KUKA KRL data list: Inconel_dataset.dat

&ACCESS RVP1
&REL 1217
&PARAM WOPTRAJECTORYID = 2
&PARAM WOPTEMPLATENAME = WopCoreTemplatePath
&PARAM DISKPATH = KRC:\R1\Program\Working Paths
DEFDAT  Inconel_dataset
;FOLD EXTERNAL DECLARATIONS;%{PE}%MKUKATPBASIS,%CEXT,%VCOMMON,%P
;FOLD BASISTECH EXT;%{PE}%MKUKATPBASIS,%CEXT,%VEXT,%P
EXT  BAS (BAS_COMMAND  :IN,REAL  :IN )
DECL INT SUCCESS
;ENDFOLD (BASISTECH EXT)
;FOLD USER EXT;%{E}%MKUKATPUSER,%CEXT,%VEXT,%P
;Make your modifications here

;ENDFOLD (USER EXT)
;ENDFOLD (EXTERNAL DECLARATIONS)

INT APP_GENNUMBER = 215375
INT APP_ANSWER
INT APP_OFFSET
DECL STATE_T APP_STATE

DECL PDAT PPDATP0={VEL 100,ACC 100,APO_DIST 5,APO_MODE #CDIS,GEAR_JERK 100.0,EXAX_IGN 0}
DECL FDAT FP0={TOOL_NO 2,BASE_NO 10,IPO_FRAME #BASE,POINT2[] " ",TQ_STATE FALSE}
DECL E6AXIS XP0={A1 -1000.000,A2 -90.000,A3 90.000,A4 0.000,A5 -90.000,A6 0.000,E1 0.000,E2 -41.000,E3 33.000,E4 0.000,E5 0.000,E6 0.000}

; Data for Routine_0
DECL LDAT LCPDATP1={VEL 1.0,ACC 100,APO_DIST 5,APO_FAC 50.0,ORI_TYP #VAR,CIRC_TYP #BASE,JERK_FAC 50.0}
DECL FDAT FP1={TOOL_NO 2,BASE_NO 10,IPO_FRAME #BASE,POINT2[] " ",TQ_STATE FALSE}
DECL E6POS XP1={X 100.000,Y 0.000,Z -100.000,A 0.000,B 0.000,C 0.000}
DECL LDAT LCPDATP2={VEL 0.116,ACC 100,APO_DIST 5,APO_FAC 50.0,ORI_TYP #VAR,CIRC_TYP #BASE,JERK_FAC 50.0}
DECL FDAT FP2={TOOL_NO 2,BASE_NO 10,IPO_FRAME #BASE,POINT2[] " ",TQ_STATE FALSE}
DECL E6POS XP2={X 50.000,Y -5.730,Z -30.020,A 0.000,B 0.000,C -28.000}
DECL LDAT LCPDATP3={VEL 0.116,ACC 100,APO_DIST 5,APO_FAC 50.0,ORI_TYP #VAR,CIRC_TYP #BASE,JERK_FAC 50.0}
DECL FDAT FP3={TOOL_NO 2,BASE_NO 10,IPO_FRAME #BASE,POINT2[] " ",TQ_STATE FALSE}
DECL E6POS XP3={X 0.000,Y -5.730,Z -30.020,A 0.000,B 0.000,C -28.000}
DECL LDAT LCPDATP4={VEL 0.116,ACC 100,APO_DIST 5,APO_FAC 50.0,ORI_TYP #VAR,CIRC_TYP #BASE,JERK_FAC 50.0}
DECL FDAT FP4={TOOL_NO 2,BASE_NO 10,IPO_FRAME #BASE,POINT2[] " ",TQ_STATE FALSE}
DECL E6POS XP4={X -50.000,Y -5.730,Z -30.020,A 0.000,B 0.000,C -28.000}
DECL LDAT LCPDATP5={VEL 0.116,ACC 100,APO_DIST 5,APO_FAC 50.0,ORI_TYP #VAR,CIRC_TYP #BASE,JERK_FAC 50.0}
DECL FDAT FP5={TOOL_NO 2,BASE_NO 10,IPO_FRAME #BASE,POINT2[] " ",TQ_STATE FALSE}
DECL E6POS XP5={X -100.000,Y -5.730,Z -30.020,A 0.000,B 0.000,C -28.000}
DECL LDAT LCPDATP6={VEL 0.099,ACC 100,APO_DIST 5,APO_FAC 50.0,ORI_TYP #VAR,CIRC_TYP #BASE,JERK_FAC 50.0}
DECL FDAT FP6={TOOL_NO 2,BASE_NO 10,IPO_FRAME #BASE,POINT2[] " ",TQ_STATE FALSE}
DECL E6POS XP6={X -100.000,Y 4.550,Z -24.510,A 0.000,B 0.000,C -40.000}
DECL LDAT LCPDATP7={VEL 0.099,ACC 100,APO_DIST 5,APO_FAC 50.0,ORI_TYP #VAR,CIRC_TYP #BASE,JERK_FAC 50.0}
DECL FDAT FP7={TOOL_NO 2,BASE_NO 10,IPO_FRAME #BASE,POINT2[] " ",TQ_STATE FALSE}
DECL E6POS XP7={X -50.000,Y 4.550,Z -24.510,A 0.000,B 0.000,C -40.000}
DECL LDAT LCPDATP8={VEL 0.099,ACC 100,APO_DIST 5,APO_FAC 50.0,ORI_TYP #VAR,CIRC_TYP #BASE,JERK_FAC 50.0}
DECL FDAT FP8={TOOL_NO 2,BASE_NO 10,IPO_FRAME #BASE,POINT2[] " ",TQ_STATE FALSE}
DECL E6POS XP8={X -0.000,Y 4.550,Z -24.510,A 0.000,B 0.000,C -40.000}
DECL LDAT LCPDATP9={VEL 0.099,ACC 100,APO_DIST 5,APO_FAC 50.0,ORI_TYP #VAR,CIRC_TYP #BASE,JERK_FAC 50.0}
DECL FDAT FP9={TOOL_NO 2,BASE_NO 10,IPO_FRAME #BASE,POINT2[] " ",TQ_STATE FALSE}
DECL E6POS XP9={X 50.000,Y 4.550,Z -24.510,A 0.000,B 0.000,C -40.000}
DECL LDAT LCPDATP10={VEL 0.075,ACC 100,APO_DIST 5,APO_FAC 50.0,ORI_TYP #VAR,CIRC_TYP #BASE,JERK_FAC 50.0}
DECL FDAT FP10={TOOL_NO 2,BASE_NO 10,IPO_FRAME #BASE,POINT2[] " ",TQ_STATE FALSE}
DECL E6POS XP10={X 50.000,Y 24.940,Z -36.820,A 0.000,B 0.000,C -23.000}
DECL LDAT LCPDATP11={VEL 0.075,ACC 100,APO_DIST 5,APO_FAC 50.0,ORI_TYP #VAR,CIRC_TYP #BASE,JERK_FAC 50.0}
DECL FDAT FP11={TOOL_NO 2,BASE_NO 10,IPO_FRAME #BASE,POINT2[] " ",TQ_STATE FALSE}
DECL E6POS XP11={X -0.000,Y 24.940,Z -36.820,A 0.000,B 0.000,C -23.000}
DECL LDAT LCPDATP12={VEL 0.075,ACC 100,APO_DIST 5,APO_FAC 50.0,ORI_TYP #VAR,CIRC_TYP #BASE,JERK_FAC 50.0}
DECL FDAT FP12={TOOL_NO 2,BASE_NO 10,IPO_FRAME #BASE,POINT2[] " ",TQ_STATE FALSE}
DECL E6POS XP12={X -50.000,Y 24.940,Z -36.820,A 0.000,B 0.000,C -23.000}
DECL LDAT LCPDATP13={VEL 0.075,ACC 100,APO_DIST 5,APO_FAC 50.0,ORI_TYP #VAR,CIRC_TYP #BASE,JERK_FAC 50.0}
DECL FDAT FP13={TOOL_NO 2,BASE_NO 10,IPO_FRAME #BASE,POINT2[] " ",TQ_STATE FALSE}
DECL E6POS XP13={X -100.000,Y 24.940,Z -36.820,A 0.000,B 0.000,C -23.000}
DECL LDAT LCPDATP14={VEL 0.113,ACC 100,APO_DIST 5,APO_FAC 50.0,ORI_TYP #VAR,CIRC_TYP #BASE,JERK_FAC 50.0}
DECL FDAT FP14={TOOL_NO 2,BASE_NO 10,IPO_FRAME #BASE,POINT2[] " ",TQ_STATE FALSE}
DECL E6POS XP14={X -100.000,Y 52.180,Z -87.790,A 0.000,B 0.000,C -4.000}
DECL LDAT LCPDATP15={VEL 0.113,ACC 100,APO_DIST 5,APO_FAC 50.0,ORI_TYP #VAR,CIRC_TYP #BASE,JERK_FAC 50.0}
DECL FDAT FP15={TOOL_NO 2,BASE_NO 10,IPO_FRAME #BASE,POINT2[] " ",TQ_STATE FALSE}
DECL E6POS XP15={X -50.000,Y 52.180,Z -87.790,A 0.000,B 0.000,C -4.000}
DECL LDAT LCPDATP16={VEL 0.113,ACC 100,APO_DIST 5,APO_FAC 50.0,ORI_TYP #VAR,CIRC_TYP #BASE,JERK_FAC 50.0}
DECL FDAT FP16={TOOL_NO 2,BASE_NO 10,IPO_FRAME #BASE,POINT2[] " ",TQ_STATE FALSE}
DECL E6POS XP16={X -0.000,Y 52.180,Z -87.790,A 0.000,B 0.000,C -4.000}
DECL LDAT LCPDATP17={VEL 0.113,ACC 100,APO_DIST 5,APO_FAC 50.0,ORI_TYP #VAR,CIRC_TYP #BASE,JERK_FAC 50.0}
DECL FDAT FP17={TOOL_NO 2,BASE_NO 10,IPO_FRAME #BASE,POINT2[] " ",TQ_STATE FALSE}
DECL E6POS XP17={X 50.000,Y 52.180,Z -87.790,A 0.000,B 0.000,C -4.000}
DECL LDAT LCPDATP18={VEL 0.086,ACC 100,APO_DIST 5,APO_FAC 50.0,ORI_TYP #VAR,CIRC_TYP #BASE,JERK_FAC 50.0}
DECL FDAT FP18={TOOL_NO 2,BASE_NO 10,IPO_FRAME #BASE,POINT2[] " ",TQ_STATE FALSE}
DECL E6POS XP18={X 50.000,Y 68.620,Z -69.900,A 0.000,B 0.000,C -3.000}
DECL LDAT LCPDATP19={VEL 0.086,ACC 100,APO_DIST 5,APO_FAC 50.0,ORI_TYP #VAR,CIRC_TYP #BASE,JERK_FAC 50.0}
DECL FDAT FP19={TOOL_NO 2,BASE_NO 10,IPO_FRAME #BASE,POINT2[] " ",TQ_STATE FALSE}
DECL E6POS XP19={X -0.000,Y 68.620,Z -69.900,A 0.000,B 0.000,C -3.000}
DECL LDAT LCPDATP20={VEL 0.086,ACC 100,APO_DIST 5,APO_FAC 50.0,ORI_TYP #VAR,CIRC_TYP #BASE,JERK_FAC 50.0}
DECL FDAT FP20={TOOL_NO 2,BASE_NO 10,IPO_FRAME #BASE,POINT2[] " ",TQ_STATE FALSE}
DECL E6POS XP20={X -50.000,Y 68.620,Z -69.900,A 0.000,B 0.000,C -3.000}
DECL LDAT LCPDATP21={VEL 0.086,ACC 100,APO_DIST 5,APO_FAC 50.0,ORI_TYP #VAR,CIRC_TYP #BASE,JERK_FAC 50.0}
DECL FDAT FP21={TOOL_NO 2,BASE_NO 10,IPO_FRAME #BASE,POINT2[] " ",TQ_STATE FALSE}
DECL E6POS XP21={X -100.000,Y 68.620,Z -69.900,A 0.000,B 0.000,C -3.000}
DECL LDAT LCPDATP22={VEL 0.073,ACC 100,APO_DIST 5,APO_FAC 50.0,ORI_TYP #VAR,CIRC_TYP #BASE,JERK_FAC 50.0}
DECL FDAT FP22={TOOL_NO 2,BASE_NO 10,IPO_FRAME #BASE,POINT2[] " ",TQ_STATE FALSE}
DECL E6POS XP22={X -100.000,Y 65.180,Z -95.090,A 0.000,B 0.000,C -14.000}
DECL LDAT LCPDATP23={VEL 0.073,ACC 100,APO_DIST 5,APO_FAC 50.0,ORI_TYP #VAR,CIRC_TYP #BASE,JERK_FAC 50.0}
DECL FDAT FP23={TOOL_NO 2,BASE_NO 10,IPO_FRAME #BASE,POINT2[] " ",TQ_STATE FALSE}
DECL E6POS XP23={X -50.000,Y 65.180,Z -95.090,A 0.000,B 0.000,C -14.000}
DECL LDAT LCPDATP24={VEL 0.073,ACC 100,APO_DIST 5,APO_FAC 50.0,ORI_TYP #VAR,CIRC_TYP #BASE,JERK_FAC 50.0}
DECL FDAT FP24={TOOL_NO 2,BASE_NO 10,IPO_FRAME #BASE,POINT2[] " ",TQ_STATE FALSE}
DECL E6POS XP24={X -0.000,Y 65.180,Z -95.090,A 0.000,B 0.000,C -14.000}
DECL LDAT LCPDATP25={VEL 0.073,ACC 100,APO_DIST 5,APO_FAC 50.0,ORI_TYP #VAR,CIRC_TYP #BASE,JERK_FAC 50.0}
DECL FDAT FP25={TOOL_NO 2,BASE_NO 10,IPO_FRAME #BASE,POINT2[] " ",TQ_STATE FALSE}
DECL E6POS XP25={X 50.000,Y 65.180,Z -95.090,A 0.000,B 0.000,C -14.000}
DECL LDAT LCPDATP26={VEL 0.137,ACC 100,APO_DIST 5,APO_FAC 50.0,ORI_TYP #VAR,CIRC_TYP #BASE,JERK_FAC 50.0}
DECL FDAT FP26={TOOL_NO 2,BASE_NO 10,IPO_FRAME #BASE,POINT2[] " ",TQ_STATE FALSE}
DECL E6POS XP26={X 50.000,Y 48.190,Z -79.460,A 0.000,B 0.000,C -35.000}
DECL LDAT LCPDATP27={VEL 0.137,ACC 100,APO_DIST 5,APO_FAC 50.0,ORI_TYP #VAR,CIRC_TYP #BASE,JERK_FAC 50.0}
DECL FDAT FP27={TOOL_NO 2,BASE_NO 10,IPO_FRAME #BASE,POINT2[] " ",TQ_STATE FALSE}
DECL E6POS XP27={X -0.000,Y 48.190,Z -79.460,A 0.000,B 0.000,C -35.000}
DECL LDAT LCPDATP28={VEL 0.137,ACC 100,APO_DIST 5,APO_FAC 50.0,ORI_TYP #VAR,CIRC_TYP #BASE,JERK_FAC 50.0}
DECL FDAT FP28={TOOL_NO 2,BASE_NO 10,IPO_FRAME #BASE,POINT2[] " ",TQ_STATE FALSE}
DECL E6POS XP28={X -50.000,Y 48.190,Z -79.460,A 0.000,B 0.000,C -35.000}
DECL LDAT LCPDATP29={VEL 0.137,ACC 100,APO_DIST 5,APO_FAC 50.0,ORI_TYP #VAR,CIRC_TYP #BASE,JERK_FAC 50.0}
DECL FDAT FP29={TOOL_NO 2,BASE_NO 10,IPO_FRAME #BASE,POINT2[] " ",TQ_STATE FALSE}
DECL E6POS XP29={X -100.000,Y 48.190,Z -79.460,A 0.000,B 0.000,C -35.000}
DECL LDAT LCPDATP30={VEL 0.082,ACC 100,APO_DIST 5,APO_FAC 50.0,ORI_TYP #VAR,CIRC_TYP #BASE,JERK_FAC 50.0}
DECL FDAT FP30={TOOL_NO 2,BASE_NO 10,IPO_FRAME #BASE,POINT2[] " ",TQ_STATE FALSE}
DECL E6POS XP30={X -100.000,Y 87.280,Z -46.640,A 0.000,B 0.000,C -32.000}
DECL LDAT LCPDATP31={VEL 0.082,ACC 100,APO_DIST 5,APO_FAC 50.0,ORI_TYP #VAR,CIRC_TYP #BASE,JERK_FAC 50.0}
DECL FDAT FP31={TOOL_NO 2,BASE_NO 10,IPO_FRAME #BASE,POINT2[] " ",TQ_STATE FALSE}
DECL E6POS XP31={X -50.000,Y 87.280,Z -46.640,A 0.000,B 0.000,C -32.000}
DECL LDAT LCPDATP32={VEL 0.082,ACC 100,APO_DIST 5,APO_FAC 50.0,ORI_TYP #VAR,CIRC_TYP #BASE,JERK_FAC 50.0}
DECL FDAT FP32={TOOL_NO 2,BASE_NO 10,IPO_FRAME #BASE,POINT2[] " ",TQ_STATE FALSE}
DECL E6POS XP32={X -0.000,Y 87.280,Z -46.640,A 0.000,B 0.000,C -32.000}
DECL LDAT LCPDATP33={VEL 0.082,ACC 100,APO_DIST 5,APO_FAC 50.0,ORI_TYP #VAR,CIRC_TYP #BASE,JERK_FAC 50.0}
DECL FDAT FP33={TOOL_NO 2,BASE_NO 10,IPO_FRAME #BASE,POINT2[] " ",TQ_STATE FALSE}
DECL E6POS XP33={X 50.000,Y 87.280,Z -46.640,A 0.000,B 0.000,C -32.000}
DECL LDAT LCPDATP34={VEL 0.086,ACC 100,APO_DIST 5,APO_FAC 50.0,ORI_TYP #VAR,CIRC_TYP #BASE,JERK_FAC 50.0}
DECL FDAT FP34={TOOL_NO 2,BASE_NO 10,IPO_FRAME #BASE,POINT2[] " ",TQ_STATE FALSE}
DECL E6POS XP34={X 50.000,Y 101.710,Z -93.610,A 0.000,B 0.000,C -19.000}
DECL LDAT LCPDATP35={VEL 0.086,ACC 100,APO_DIST 5,APO_FAC 50.0,ORI_TYP #VAR,CIRC_TYP #BASE,JERK_FAC 50.0}
DECL FDAT FP35={TOOL_NO 2,BASE_NO 10,IPO_FRAME #BASE,POINT2[] " ",TQ_STATE FALSE}
DECL E6POS XP35={X -0.000,Y 101.710,Z -93.610,A 0.000,B 0.000,C -19.000}
DECL LDAT LCPDATP36={VEL 0.086,ACC 100,APO_DIST 5,APO_FAC 50.0,ORI_TYP #VAR,CIRC_TYP #BASE,JERK_FAC 50.0}
DECL FDAT FP36={TOOL_NO 2,BASE_NO 10,IPO_FRAME #BASE,POINT2[] " ",TQ_STATE FALSE}
DECL E6POS XP36={X -50.000,Y 101.710,Z -93.610,A 0.000,B 0.000,C -19.000}
DECL LDAT LCPDATP37={VEL 0.086,ACC 100,APO_DIST 5,APO_FAC 50.0,ORI_TYP #VAR,CIRC_TYP #BASE,JERK_FAC 50.0}
DECL FDAT FP37={TOOL_NO 2,BASE_NO 10,IPO_FRAME #BASE,POINT2[] " ",TQ_STATE FALSE}
DECL E6POS XP37={X -100.000,Y 101.710,Z -93.610,A 0.000,B 0.000,C -19.000}
DECL LDAT LCPDATP38={VEL 0.097,ACC 100,APO_DIST 5,APO_FAC 50.0,ORI_TYP #VAR,CIRC_TYP #BASE,JERK_FAC 50.0}
DECL FDAT FP38={TOOL_NO 2,BASE_NO 10,IPO_FRAME #BASE,POINT2[] " ",TQ_STATE FALSE}
DECL E6POS XP38={X -100.000,Y 117.680,Z -79.350,A 0.000,B 0.000,C -21.000}
DECL LDAT LCPDATP39={VEL 0.097,ACC 100,APO_DIST 5,APO_FAC 50.0,ORI_TYP #VAR,CIRC_TYP #BASE,JERK_FAC 50.0}
DECL FDAT FP39={TOOL_NO 2,BASE_NO 10,IPO_FRAME #BASE,POINT2[] " ",TQ_STATE FALSE}
DECL E6POS XP39={X -50.000,Y 117.680,Z -79.350,A 0.000,B 0.000,C -21.000}
DECL LDAT LCPDATP40={VEL 0.097,ACC 100,APO_DIST 5,APO_FAC 50.0,ORI_TYP #VAR,CIRC_TYP #BASE,JERK_FAC 50.0}
DECL FDAT FP40={TOOL_NO 2,BASE_NO 10,IPO_FRAME #BASE,POINT2[] " ",TQ_STATE FALSE}
DECL E6POS XP40={X -0.000,Y 117.680,Z -79.350,A 0.000,B 0.000,C -21.000}
DECL LDAT LCPDATP41={VEL 0.097,ACC 100,APO_DIST 5,APO_FAC 50.0,ORI_TYP #VAR,CIRC_TYP #BASE,JERK_FAC 50.0}
DECL FDAT FP41={TOOL_NO 2,BASE_NO 10,IPO_FRAME #BASE,POINT2[] " ",TQ_STATE FALSE}
DECL E6POS XP41={X 50.000,Y 117.680,Z -79.350,A 0.000,B 0.000,C -21.000}
DECL LDAT LCPDATP42={VEL 0.136,ACC 100,APO_DIST 5,APO_FAC 50.0,ORI_TYP #VAR,CIRC_TYP #BASE,JERK_FAC 50.0}
DECL FDAT FP42={TOOL_NO 2,BASE_NO 10,IPO_FRAME #BASE,POINT2[] " ",TQ_STATE FALSE}
DECL E6POS XP42={X 50.000,Y 150.480,Z -65.980,A 0.000,B 0.000,C -10.000}
DECL LDAT LCPDATP43={VEL 0.136,ACC 100,APO_DIST 5,APO_FAC 50.0,ORI_TYP #VAR,CIRC_TYP #BASE,JERK_FAC 50.0}
DECL FDAT FP43={TOOL_NO 2,BASE_NO 10,IPO_FRAME #BASE,POINT2[] " ",TQ_STATE FALSE}
DECL E6POS XP43={X -0.000,Y 150.480,Z -65.980,A 0.000,B 0.000,C -10.000}
DECL LDAT LCPDATP44={VEL 0.136,ACC 100,APO_DIST 5,APO_FAC 50.0,ORI_TYP #VAR,CIRC_TYP #BASE,JERK_FAC 50.0}
DECL FDAT FP44={TOOL_NO 2,BASE_NO 10,IPO_FRAME #BASE,POINT2[] " ",TQ_STATE FALSE}
DECL E6POS XP44={X -50.000,Y 150.480,Z -65.980,A 0.000,B 0.000,C -10.000}
DECL LDAT LCPDATP45={VEL 0.136,ACC 100,APO_DIST 5,APO_FAC 50.0,ORI_TYP #VAR,CIRC_TYP #BASE,JERK_FAC 50.0}
DECL FDAT FP45={TOOL_NO 2,BASE_NO 10,IPO_FRAME #BASE,POINT2[] " ",TQ_STATE FALSE}
DECL E6POS XP45={X -100.000,Y 150.480,Z -65.980,A 0.000,B 0.000,C -10.000}
DECL LDAT LCPDATP46={VEL 0.107,ACC 100,APO_DIST 5,APO_FAC 50.0,ORI_TYP #VAR,CIRC_TYP #BASE,JERK_FAC 50.0}
DECL FDAT FP46={TOOL_NO 2,BASE_NO 10,IPO_FRAME #BASE,POINT2[] " ",TQ_STATE FALSE}
DECL E6POS XP46={X -100.000,Y 132.510,Z -57.520,A 0.000,B 0.000,C -38.000}
DECL LDAT LCPDATP47={VEL 0.107,ACC 100,APO_DIST 5,APO_FAC 50.0,ORI_TYP #VAR,CIRC_TYP #BASE,JERK_FAC 50.0}
DECL FDAT FP47={TOOL_NO 2,BASE_NO 10,IPO_FRAME #BASE,POINT2[] " ",TQ_STATE FALSE}
DECL E6POS XP47={X -50.000,Y 132.510,Z -57.520,A 0.000,B 0.000,C -38.000}
DECL LDAT LCPDATP48={VEL 0.107,ACC 100,APO_DIST 5,APO_FAC 50.0,ORI_TYP #VAR,CIRC_TYP #BASE,JERK_FAC 50.0}
DECL FDAT FP48={TOOL_NO 2,BASE_NO 10,IPO_FRAME #BASE,POINT2[] " ",TQ_STATE FALSE}
DECL E6POS XP48={X -0.000,Y 132.510,Z -57.520,A 0.000,B 0.000,C -38.000}
DECL LDAT LCPDATP49={VEL 0.107,ACC 100,APO_DIST 5,APO_FAC 50.0,ORI_TYP #VAR,CIRC_TYP #BASE,JERK_FAC 50.0}
DECL FDAT FP49={TOOL_NO 2,BASE_NO 10,IPO_FRAME #BASE,POINT2[] " ",TQ_STATE FALSE}
DECL E6POS XP49={X 50.000,Y 132.510,Z -57.520,A 0.000,B 0.000,C -38.000}
DECL LDAT LCPDATP50={VEL 0.09,ACC 100,APO_DIST 5,APO_FAC 50.0,ORI_TYP #VAR,CIRC_TYP #BASE,JERK_FAC 50.0}
DECL FDAT FP50={TOOL_NO 2,BASE_NO 10,IPO_FRAME #BASE,POINT2[] " ",TQ_STATE FALSE}
DECL E6POS XP50={X 50.000,Y 148.310,Z -68.770,A 0.000,B 0.000,C -33.000}
DECL LDAT LCPDATP51={VEL 0.09,ACC 100,APO_DIST 5,APO_FAC 50.0,ORI_TYP #VAR,CIRC_TYP #BASE,JERK_FAC 50.0}
DECL FDAT FP51={TOOL_NO 2,BASE_NO 10,IPO_FRAME #BASE,POINT2[] " ",TQ_STATE FALSE}
DECL E6POS XP51={X -0.000,Y 148.310,Z -68.770,A 0.000,B 0.000,C -33.000}
DECL LDAT LCPDATP52={VEL 0.09,ACC 100,APO_DIST 5,APO_FAC 50.0,ORI_TYP #VAR,CIRC_TYP #BASE,JERK_FAC 50.0}
DECL FDAT FP52={TOOL_NO 2,BASE_NO 10,IPO_FRAME #BASE,POINT2[] " ",TQ_STATE FALSE}
DECL E6POS XP52={X -50.000,Y 148.310,Z -68.770,A 0.000,B 0.000,C -33.000}
DECL LDAT LCPDATP53={VEL 0.09,ACC 100,APO_DIST 5,APO_FAC 50.0,ORI_TYP #VAR,CIRC_TYP #BASE,JERK_FAC 50.0}
DECL FDAT FP53={TOOL_NO 2,BASE_NO 10,IPO_FRAME #BASE,POINT2[] " ",TQ_STATE FALSE}
DECL E6POS XP53={X -100.000,Y 148.310,Z -68.770,A 0.000,B 0.000,C -33.000}
DECL LDAT LCPDATP54={VEL 0.132,ACC 100,APO_DIST 5,APO_FAC 50.0,ORI_TYP #VAR,CIRC_TYP #BASE,JERK_FAC 50.0}
DECL FDAT FP54={TOOL_NO 2,BASE_NO 10,IPO_FRAME #BASE,POINT2[] " ",TQ_STATE FALSE}
DECL E6POS XP54={X -100.000,Y 203.750,Z -95.870,A 0.000,B 0.000,C -3.000}
DECL LDAT LCPDATP55={VEL 0.132,ACC 100,APO_DIST 5,APO_FAC 50.0,ORI_TYP #VAR,CIRC_TYP #BASE,JERK_FAC 50.0}
DECL FDAT FP55={TOOL_NO 2,BASE_NO 10,IPO_FRAME #BASE,POINT2[] " ",TQ_STATE FALSE}
DECL E6POS XP55={X -50.000,Y 203.750,Z -95.870,A 0.000,B 0.000,C -3.000}
DECL LDAT LCPDATP56={VEL 0.132,ACC 100,APO_DIST 5,APO_FAC 50.0,ORI_TYP #VAR,CIRC_TYP #BASE,JERK_FAC 50.0}
DECL FDAT FP56={TOOL_NO 2,BASE_NO 10,IPO_FRAME #BASE,POINT2[] " ",TQ_STATE FALSE}
DECL E6POS XP56={X -0.000,Y 203.750,Z -95.870,A 0.000,B 0.000,C -3.000}
DECL LDAT LCPDATP57={VEL 0.132,ACC 100,APO_DIST 5,APO_FAC 50.0,ORI_TYP #VAR,CIRC_TYP #BASE,JERK_FAC 50.0}
DECL FDAT FP57={TOOL_NO 2,BASE_NO 10,IPO_FRAME #BASE,POINT2[] " ",TQ_STATE FALSE}
DECL E6POS XP57={X 50.000,Y 203.750,Z -95.870,A 0.000,B 0.000,C -3.000}
DECL LDAT LCPDATP58={VEL 0.068,ACC 100,APO_DIST 5,APO_FAC 50.0,ORI_TYP #VAR,CIRC_TYP #BASE,JERK_FAC 50.0}
DECL FDAT FP58={TOOL_NO 2,BASE_NO 10,IPO_FRAME #BASE,POINT2[] " ",TQ_STATE FALSE}
DECL E6POS XP58={X 50.000,Y 221.500,Z -80.990,A 0.000,B 0.000,C -1.000}
DECL LDAT LCPDATP59={VEL 0.068,ACC 100,APO_DIST 5,APO_FAC 50.0,ORI_TYP #VAR,CIRC_TYP #BASE,JERK_FAC 50.0}
DECL FDAT FP59={TOOL_NO 2,BASE_NO 10,IPO_FRAME #BASE,POINT2[] " ",TQ_STATE FALSE}
DECL E6POS XP59={X -0.000,Y 221.500,Z -80.990,A 0.000,B 0.000,C -1.000}
DECL LDAT LCPDATP60={VEL 0.068,ACC 100,APO_DIST 5,APO_FAC 50.0,ORI_TYP #VAR,CIRC_TYP #BASE,JERK_FAC 50.0}
DECL FDAT FP60={TOOL_NO 2,BASE_NO 10,IPO_FRAME #BASE,POINT2[] " ",TQ_STATE FALSE}
DECL E6POS XP60={X -50.000,Y 221.500,Z -80.990,A 0.000,B 0.000,C -1.000}
DECL LDAT LCPDATP61={VEL 0.068,ACC 100,APO_DIST 5,APO_FAC 50.0,ORI_TYP #VAR,CIRC_TYP #BASE,JERK_FAC 50.0}
DECL FDAT FP61={TOOL_NO 2,BASE_NO 10,IPO_FRAME #BASE,POINT2[] " ",TQ_STATE FALSE}
DECL E6POS XP61={X -100.000,Y 221.500,Z -80.990,A 0.000,B 0.000,C -1.000}
DECL LDAT LCPDATP62={VEL 0.115,ACC 100,APO_DIST 5,APO_FAC 50.0,ORI_TYP #VAR,CIRC_TYP #BASE,JERK_FAC 50.0}
DECL FDAT FP62={TOOL_NO 2,BASE_NO 10,IPO_FRAME #BASE,POINT2[] " ",TQ_STATE FALSE}
DECL E6POS XP62={X -100.000,Y 206.270,Z -52.830,A 0.000,B 0.000,C -30.000}
DECL LDAT LCPDATP63={VEL 0.115,ACC 100,APO_DIST 5,APO_FAC 50.0,ORI_TYP #VAR,CIRC_TYP #BASE,JERK_FAC 50.0}
DECL FDAT FP63={TOOL_NO 2,BASE_NO 10,IPO_FRAME #BASE,POINT2[] " ",TQ_STATE FALSE}
DECL E6POS XP63={X -50.000,Y 206.270,Z -52.830,A 0.000,B 0.000,C -30.000}
DECL LDAT LCPDATP64={VEL 0.115,ACC 100,APO_DIST 5,APO_FAC 50.0,ORI_TYP #VAR,CIRC_TYP #BASE,JERK_FAC 50.0}
DECL FDAT FP64={TOOL_NO 2,BASE_NO 10,IPO_FRAME #BASE,POINT2[] " ",TQ_STATE FALSE}
DECL E6POS XP64={X -0.000,Y 206.270,Z -52.830,A 0.000,B 0.000,C -30.000}
DECL LDAT LCPDATP65={VEL 0.115,ACC 100,APO_DIST 5,APO_FAC 50.0,ORI_TYP #VAR,CIRC_TYP #BASE,JERK_FAC 50.0}
DECL FDAT FP65={TOOL_NO 2,BASE_NO 10,IPO_FRAME #BASE,POINT2[] " ",TQ_STATE FALSE}
DECL E6POS XP65={X 50.000,Y 206.270,Z -52.830,A 0.000,B 0.000,C -30.000}
DECL LDAT LCPDATP66={VEL 0.111,ACC 100,APO_DIST 5,APO_FAC 50.0,ORI_TYP #VAR,CIRC_TYP #BASE,JERK_FAC 50.0}
DECL FDAT FP66={TOOL_NO 2,BASE_NO 10,IPO_FRAME #BASE,POINT2[] " ",TQ_STATE FALSE}
DECL E6POS XP66={X 50.000,Y 214.030,Z -89.530,A 0.000,B 0.000,C -24.000}
DECL LDAT LCPDATP67={VEL 0.111,ACC 100,APO_DIST 5,APO_FAC 50.0,ORI_TYP #VAR,CIRC_TYP #BASE,JERK_FAC 50.0}
DECL FDAT FP67={TOOL_NO 2,BASE_NO 10,IPO_FRAME #BASE,POINT2[] " ",TQ_STATE FALSE}
DECL E6POS XP67={X -0.000,Y 214.030,Z -89.530,A 0.000,B 0.000,C -24.000}
DECL LDAT LCPDATP68={VEL 0.111,ACC 100,APO_DIST 5,APO_FAC 50.0,ORI_TYP #VAR,CIRC_TYP #BASE,JERK_FAC 50.0}
DECL FDAT FP68={TOOL_NO 2,BASE_NO 10,IPO_FRAME #BASE,POINT2[] " ",TQ_STATE FALSE}
DECL E6POS XP68={X -50.000,Y 214.030,Z -89.530,A 0.000,B 0.000,C -24.000}
DECL LDAT LCPDATP69={VEL 0.111,ACC 100,APO_DIST 5,APO_FAC 50.0,ORI_TYP #VAR,CIRC_TYP #BASE,JERK_FAC 50.0}
DECL FDAT FP69={TOOL_NO 2,BASE_NO 10,IPO_FRAME #BASE,POINT2[] " ",TQ_STATE FALSE}
DECL E6POS XP69={X -100.000,Y 214.030,Z -89.530,A 0.000,B 0.000,C -24.000}
DECL LDAT LCPDATP70={VEL 0.124,ACC 100,APO_DIST 5,APO_FAC 50.0,ORI_TYP #VAR,CIRC_TYP #BASE,JERK_FAC 50.0}
DECL FDAT FP70={TOOL_NO 2,BASE_NO 10,IPO_FRAME #BASE,POINT2[] " ",TQ_STATE FALSE}
DECL E6POS XP70={X -100.000,Y 264.220,Z -41.970,A 0.000,B 0.000,C -2.000}
DECL LDAT LCPDATP71={VEL 0.124,ACC 100,APO_DIST 5,APO_FAC 50.0,ORI_TYP #VAR,CIRC_TYP #BASE,JERK_FAC 50.0}
DECL FDAT FP71={TOOL_NO 2,BASE_NO 10,IPO_FRAME #BASE,POINT2[] " ",TQ_STATE FALSE}
DECL E6POS XP71={X -50.000,Y 264.220,Z -41.970,A 0.000,B 0.000,C -2.000}
DECL LDAT LCPDATP72={VEL 0.124,ACC 100,APO_DIST 5,APO_FAC 50.0,ORI_TYP #VAR,CIRC_TYP #BASE,JERK_FAC 50.0}
DECL FDAT FP72={TOOL_NO 2,BASE_NO 10,IPO_FRAME #BASE,POINT2[] " ",TQ_STATE FALSE}
DECL E6POS XP72={X -0.000,Y 264.220,Z -41.970,A 0.000,B 0.000,C -2.000}
DECL LDAT LCPDATP73={VEL 0.124,ACC 100,APO_DIST 5,APO_FAC 50.0,ORI_TYP #VAR,CIRC_TYP #BASE,JERK_FAC 50.0}
DECL FDAT FP73={TOOL_NO 2,BASE_NO 10,IPO_FRAME #BASE,POINT2[] " ",TQ_STATE FALSE}
DECL E6POS XP73={X 50.000,Y 264.220,Z -41.970,A 0.000,B 0.000,C -2.000}
DECL LDAT LCPDATP74={VEL 0.112,ACC 100,APO_DIST 5,APO_FAC 50.0,ORI_TYP #VAR,CIRC_TYP #BASE,JERK_FAC 50.0}
DECL FDAT FP74={TOOL_NO 2,BASE_NO 10,IPO_FRAME #BASE,POINT2[] " ",TQ_STATE FALSE}
DECL E6POS XP74={X 50.000,Y 254.510,Z -62.120,A 0.000,B 0.000,C -24.000}
DECL LDAT LCPDATP75={VEL 0.112,ACC 100,APO_DIST 5,APO_FAC 50.0,ORI_TYP #VAR,CIRC_TYP #BASE,JERK_FAC 50.0}
DECL FDAT FP75={TOOL_NO 2,BASE_NO 10,IPO_FRAME #BASE,POINT2[] " ",TQ_STATE FALSE}
DECL E6POS XP75={X -0.000,Y 254.510,Z -62.120,A 0.000,B 0.000,C -24.000}
DECL LDAT LCPDATP76={VEL 0.112,ACC 100,APO_DIST 5,APO_FAC 50.0,ORI_TYP #VAR,CIRC_TYP #BASE,JERK_FAC 50.0}
DECL FDAT FP76={TOOL_NO 2,BASE_NO 10,IPO_FRAME #BASE,POINT2[] " ",TQ_STATE FALSE}
DECL E6POS XP76={X -50.000,Y 254.510,Z -62.120,A 0.000,B 0.000,C -24.000}
DECL LDAT LCPDATP77={VEL 0.112,ACC 100,APO_DIST 5,APO_FAC 50.0,ORI_TYP #VAR,CIRC_TYP #BASE,JERK_FAC 50.0}
DECL FDAT FP77={TOOL_NO 2,BASE_NO 10,IPO_FRAME #BASE,POINT2[] " ",TQ_STATE FALSE}
DECL E6POS XP77={X -100.000,Y 254.510,Z -62.120,A 0.000,B 0.000,C -24.000}
DECL LDAT LCPDATP78={VEL 0.109,ACC 100,APO_DIST 5,APO_FAC 50.0,ORI_TYP #VAR,CIRC_TYP #BASE,JERK_FAC 50.0}
DECL FDAT FP78={TOOL_NO 2,BASE_NO 10,IPO_FRAME #BASE,POINT2[] " ",TQ_STATE FALSE}
DECL E6POS XP78={X -100.000,Y 269.410,Z -36.410,A 0.000,B 0.000,C -36.000}
DECL LDAT LCPDATP79={VEL 0.109,ACC 100,APO_DIST 5,APO_FAC 50.0,ORI_TYP #VAR,CIRC_TYP #BASE,JERK_FAC 50.0}
DECL FDAT FP79={TOOL_NO 2,BASE_NO 10,IPO_FRAME #BASE,POINT2[] " ",TQ_STATE FALSE}
DECL E6POS XP79={X -50.000,Y 269.410,Z -36.410,A 0.000,B 0.000,C -36.000}
DECL LDAT LCPDATP80={VEL 0.109,ACC 100,APO_DIST 5,APO_FAC 50.0,ORI_TYP #VAR,CIRC_TYP #BASE,JERK_FAC 50.0}
DECL FDAT FP80={TOOL_NO 2,BASE_NO 10,IPO_FRAME #BASE,POINT2[] " ",TQ_STATE FALSE}
DECL E6POS XP80={X -0.000,Y 269.410,Z -36.410,A 0.000,B 0.000,C -36.000}
DECL LDAT LCPDATP81={VEL 0.109,ACC 100,APO_DIST 5,APO_FAC 50.0,ORI_TYP #VAR,CIRC_TYP #BASE,JERK_FAC 50.0}
DECL FDAT FP81={TOOL_NO 2,BASE_NO 10,IPO_FRAME #BASE,POINT2[] " ",TQ_STATE FALSE}
DECL E6POS XP81={X 50.000,Y 269.410,Z -36.410,A 0.000,B 0.000,C -36.000}
DECL LDAT LCPDATP82={VEL 0.104,ACC 100,APO_DIST 5,APO_FAC 50.0,ORI_TYP #VAR,CIRC_TYP #BASE,JERK_FAC 50.0}
DECL FDAT FP82={TOOL_NO 2,BASE_NO 10,IPO_FRAME #BASE,POINT2[] " ",TQ_STATE FALSE}
DECL E6POS XP82={X 50.000,Y 288.080,Z -43.260,A 0.000,B 0.000,C -28.000}
DECL LDAT LCPDATP83={VEL 0.104,ACC 100,APO_DIST 5,APO_FAC 50.0,ORI_TYP #VAR,CIRC_TYP #BASE,JERK_FAC 50.0}
DECL FDAT FP83={TOOL_NO 2,BASE_NO 10,IPO_FRAME #BASE,POINT2[] " ",TQ_STATE FALSE}
DECL E6POS XP83={X -0.000,Y 288.080,Z -43.260,A 0.000,B 0.000,C -28.000}
DECL LDAT LCPDATP84={VEL 0.104,ACC 100,APO_DIST 5,APO_FAC 50.0,ORI_TYP #VAR,CIRC_TYP #BASE,JERK_FAC 50.0}
DECL FDAT FP84={TOOL_NO 2,BASE_NO 10,IPO_FRAME #BASE,POINT2[] " ",TQ_STATE FALSE}
DECL E6POS XP84={X -50.000,Y 288.080,Z -43.260,A 0.000,B 0.000,C -28.000}
DECL LDAT LCPDATP85={VEL 0.104,ACC 100,APO_DIST 5,APO_FAC 50.0,ORI_TYP #VAR,CIRC_TYP #BASE,JERK_FAC 50.0}
DECL FDAT FP85={TOOL_NO 2,BASE_NO 10,IPO_FRAME #BASE,POINT2[] " ",TQ_STATE FALSE}
DECL E6POS XP85={X -100.000,Y 288.080,Z -43.260,A 0.000,B 0.000,C -28.000}
DECL LDAT LCPDATP86={VEL 0.053,ACC 100,APO_DIST 5,APO_FAC 50.0,ORI_TYP #VAR,CIRC_TYP #BASE,JERK_FAC 50.0}
DECL FDAT FP86={TOOL_NO 2,BASE_NO 10,IPO_FRAME #BASE,POINT2[] " ",TQ_STATE FALSE}
DECL E6POS XP86={X -100.000,Y 303.890,Z -73.230,A 0.000,B 0.000,C -18.000}
DECL LDAT LCPDATP87={VEL 0.053,ACC 100,APO_DIST 5,APO_FAC 50.0,ORI_TYP #VAR,CIRC_TYP #BASE,JERK_FAC 50.0}
DECL FDAT FP87={TOOL_NO 2,BASE_NO 10,IPO_FRAME #BASE,POINT2[] " ",TQ_STATE FALSE}
DECL E6POS XP87={X -50.000,Y 303.890,Z -73.230,A 0.000,B 0.000,C -18.000}
DECL LDAT LCPDATP88={VEL 0.053,ACC 100,APO_DIST 5,APO_FAC 50.0,ORI_TYP #VAR,CIRC_TYP #BASE,JERK_FAC 50.0}
DECL FDAT FP88={TOOL_NO 2,BASE_NO 10,IPO_FRAME #BASE,POINT2[] " ",TQ_STATE FALSE}
DECL E6POS XP88={X -0.000,Y 303.890,Z -73.230,A 0.000,B 0.000,C -18.000}
DECL LDAT LCPDATP89={VEL 0.053,ACC 100,APO_DIST 5,APO_FAC 50.0,ORI_TYP #VAR,CIRC_TYP #BASE,JERK_FAC 50.0}
DECL FDAT FP89={TOOL_NO 2,BASE_NO 10,IPO_FRAME #BASE,POINT2[] " ",TQ_STATE FALSE}
DECL E6POS XP89={X 50.000,Y 303.890,Z -73.230,A 0.000,B 0.000,C -18.000}
DECL LDAT LCPDATP90={VEL 0.063,ACC 100,APO_DIST 5,APO_FAC 50.0,ORI_TYP #VAR,CIRC_TYP #BASE,JERK_FAC 50.0}
DECL FDAT FP90={TOOL_NO 2,BASE_NO 10,IPO_FRAME #BASE,POINT2[] " ",TQ_STATE FALSE}
DECL E6POS XP90={X 50.000,Y 335.430,Z -94.640,A 0.000,B 0.000,C -5.000}
DECL LDAT LCPDATP91={VEL 0.063,ACC 100,APO_DIST 5,APO_FAC 50.0,ORI_TYP #VAR,CIRC_TYP #BASE,JERK_FAC 50.0}
DECL FDAT FP91={TOOL_NO 2,BASE_NO 10,IPO_FRAME #BASE,POINT2[] " ",TQ_STATE FALSE}
DECL E6POS XP91={X -0.000,Y 335.430,Z -94.640,A 0.000,B 0.000,C -5.000}
DECL LDAT LCPDATP92={VEL 0.063,ACC 100,APO_DIST 5,APO_FAC 50.0,ORI_TYP #VAR,CIRC_TYP #BASE,JERK_FAC 50.0}
DECL FDAT FP92={TOOL_NO 2,BASE_NO 10,IPO_FRAME #BASE,POINT2[] " ",TQ_STATE FALSE}
DECL E6POS XP92={X -50.000,Y 335.430,Z -94.640,A 0.000,B 0.000,C -5.000}
DECL LDAT LCPDATP93={VEL 0.063,ACC 100,APO_DIST 5,APO_FAC 50.0,ORI_TYP #VAR,CIRC_TYP #BASE,JERK_FAC 50.0}
DECL FDAT FP93={TOOL_NO 2,BASE_NO 10,IPO_FRAME #BASE,POINT2[] " ",TQ_STATE FALSE}
DECL E6POS XP93={X -100.000,Y 335.430,Z -94.640,A 0.000,B 0.000,C -5.000}
DECL LDAT LCPDATP94={VEL 0.5,ACC 100,APO_DIST 5,APO_FAC 50.0,ORI_TYP #VAR,CIRC_TYP #BASE,JERK_FAC 50.0}
DECL FDAT FP94={TOOL_NO 2,BASE_NO 10,IPO_FRAME #BASE,POINT2[] " ",TQ_STATE FALSE}
DECL E6POS XP94={X -150.000,Y 343.710,Z -50.000,A 0.000,B 0.000,C 0.000}
DECL LDAT LCPDATP95={VEL 1.0,ACC 100,APO_DIST 5,APO_FAC 50.0,ORI_TYP #VAR,CIRC_TYP #BASE,JERK_FAC 50.0}
DECL FDAT FP95={TOOL_NO 2,BASE_NO 10,IPO_FRAME #BASE,POINT2[] " ",TQ_STATE FALSE}
DECL E6POS XP95={X -150.000,Y 380.000,Z -20.000,A 0.000,B 0.000,C 0.000}
DECL LDAT LCPDATP96={VEL 1.0,ACC 100,APO_DIST 5,APO_FAC 50.0,ORI_TYP #VAR,CIRC_TYP #BASE,JERK_FAC 50.0}
DECL FDAT FP96={TOOL_NO 2,BASE_NO 10,IPO_FRAME #BASE,POINT2[] " ",TQ_STATE FALSE}
DECL E6POS XP96={X 100.000,Y 380.000,Z -20.000,A 0.000,B 0.000,C 0.000}
;ENDDAT for Routine_0


; Data for Routine_1
DECL LDAT LCPDATP97={VEL 1.0,ACC 100,APO_DIST 5,APO_FAC 50.0,ORI_TYP #VAR,CIRC_TYP #BASE,JERK_FAC 50.0}
DECL FDAT FP97={TOOL_NO 2,BASE_NO 9,IPO_FRAME #BASE,POINT2[] " ",TQ_STATE FALSE}
DECL E6POS XP97={X 100.000,Y 0.000,Z -100.000,A 0.000,B 0.000,C 0.000}
DECL LDAT LCPDATP98={VEL 0.065,ACC 100,APO_DIST 5,APO_FAC 50.0,ORI_TYP #VAR,CIRC_TYP #BASE,JERK_FAC 50.0}
DECL FDAT FP98={TOOL_NO 2,BASE_NO 9,IPO_FRAME #BASE,POINT2[] " ",TQ_STATE FALSE}
DECL E6POS XP98={X 50.000,Y -2.120,Z -67.490,A 0.000,B 0.000,C -12.000}
DECL LDAT LCPDATP99={VEL 0.065,ACC 100,APO_DIST 5,APO_FAC 50.0,ORI_TYP #VAR,CIRC_TYP #BASE,JERK_FAC 50.0}
DECL FDAT FP99={TOOL_NO 2,BASE_NO 9,IPO_FRAME #BASE,POINT2[] " ",TQ_STATE FALSE}
DECL E6POS XP99={X 0.000,Y -2.120,Z -67.490,A 0.000,B 0.000,C -12.000}
DECL LDAT LCPDATP100={VEL 0.065,ACC 100,APO_DIST 5,APO_FAC 50.0,ORI_TYP #VAR,CIRC_TYP #BASE,JERK_FAC 50.0}
DECL FDAT FP100={TOOL_NO 2,BASE_NO 9,IPO_FRAME #BASE,POINT2[] " ",TQ_STATE FALSE}
DECL E6POS XP100={X -50.000,Y -2.120,Z -67.490,A 0.000,B 0.000,C -12.000}
DECL LDAT LCPDATP101={VEL 0.065,ACC 100,APO_DIST 5,APO_FAC 50.0,ORI_TYP #VAR,CIRC_TYP #BASE,JERK_FAC 50.0}
DECL FDAT FP101={TOOL_NO 2,BASE_NO 9,IPO_FRAME #BASE,POINT2[] " ",TQ_STATE FALSE}
DECL E6POS XP101={X -100.000,Y -2.120,Z -67.490,A 0.000,B 0.000,C -12.000}
DECL LDAT LCPDATP102={VEL 0.088,ACC 100,APO_DIST 5,APO_FAC 50.0,ORI_TYP #VAR,CIRC_TYP #BASE,JERK_FAC 50.0}
DECL FDAT FP102={TOOL_NO 2,BASE_NO 9,IPO_FRAME #BASE,POINT2[] " ",TQ_STATE FALSE}
DECL E6POS XP102={X -100.000,Y 15.760,Z -30.600,A 0.000,B 0.000,C -17.000}
DECL LDAT LCPDATP103={VEL 0.088,ACC 100,APO_DIST 5,APO_FAC 50.0,ORI_TYP #VAR,CIRC_TYP #BASE,JERK_FAC 50.0}
DECL FDAT FP103={TOOL_NO 2,BASE_NO 9,IPO_FRAME #BASE,POINT2[] " ",TQ_STATE FALSE}
DECL E6POS XP103={X -50.000,Y 15.760,Z -30.600,A 0.000,B 0.000,C -17.000}
DECL LDAT LCPDATP104={VEL 0.088,ACC 100,APO_DIST 5,APO_FAC 50.0,ORI_TYP #VAR,CIRC_TYP #BASE,JERK_FAC 50.0}
DECL FDAT FP104={TOOL_NO 2,BASE_NO 9,IPO_FRAME #BASE,POINT2[] " ",TQ_STATE FALSE}
DECL E6POS XP104={X -0.000,Y 15.760,Z -30.600,A 0.000,B 0.000,C -17.000}
DECL LDAT LCPDATP105={VEL 0.088,ACC 100,APO_DIST 5,APO_FAC 50.0,ORI_TYP #VAR,CIRC_TYP #BASE,JERK_FAC 50.0}
DECL FDAT FP105={TOOL_NO 2,BASE_NO 9,IPO_FRAME #BASE,POINT2[] " ",TQ_STATE FALSE}
DECL E6POS XP105={X 50.000,Y 15.760,Z -30.600,A 0.000,B 0.000,C -17.000}
DECL LDAT LCPDATP106={VEL 0.06,ACC 100,APO_DIST 5,APO_FAC 50.0,ORI_TYP #VAR,CIRC_TYP #BASE,JERK_FAC 50.0}
DECL FDAT FP106={TOOL_NO 2,BASE_NO 9,IPO_FRAME #BASE,POINT2[] " ",TQ_STATE FALSE}
DECL E6POS XP106={X 50.000,Y 13.210,Z -73.250,A 0.000,B 0.000,C -22.000}
DECL LDAT LCPDATP107={VEL 0.06,ACC 100,APO_DIST 5,APO_FAC 50.0,ORI_TYP #VAR,CIRC_TYP #BASE,JERK_FAC 50.0}
DECL FDAT FP107={TOOL_NO 2,BASE_NO 9,IPO_FRAME #BASE,POINT2[] " ",TQ_STATE FALSE}
DECL E6POS XP107={X -0.000,Y 13.210,Z -73.250,A 0.000,B 0.000,C -22.000}
DECL LDAT LCPDATP108={VEL 0.06,ACC 100,APO_DIST 5,APO_FAC 50.0,ORI_TYP #VAR,CIRC_TYP #BASE,JERK_FAC 50.0}
DECL FDAT FP108={TOOL_NO 2,BASE_NO 9,IPO_FRAME #BASE,POINT2[] " ",TQ_STATE FALSE}
DECL E6POS XP108={X -50.000,Y 13.210,Z -73.250,A 0.000,B 0.000,C -22.000}
DECL LDAT LCPDATP109={VEL 0.06,ACC 100,APO_DIST 5,APO_FAC 50.0,ORI_TYP #VAR,CIRC_TYP #BASE,JERK_FAC 50.0}
DECL FDAT FP109={TOOL_NO 2,BASE_NO 9,IPO_FRAME #BASE,POINT2[] " ",TQ_STATE FALSE}
DECL E6POS XP109={X -100.000,Y 13.210,Z -73.250,A 0.000,B 0.000,C -22.000}
DECL LDAT LCPDATP110={VEL 0.135,ACC 100,APO_DIST 5,APO_FAC 50.0,ORI_TYP #VAR,CIRC_TYP #BASE,JERK_FAC 50.0}
DECL FDAT FP110={TOOL_NO 2,BASE_NO 9,IPO_FRAME #BASE,POINT2[] " ",TQ_STATE FALSE}
DECL E6POS XP110={X -100.000,Y 40.110,Z -53.550,A 0.000,B 0.000,C -17.000}
DECL LDAT LCPDATP111={VEL 0.135,ACC 100,APO_DIST 5,APO_FAC 50.0,ORI_TYP #VAR,CIRC_TYP #BASE,JERK_FAC 50.0}
DECL FDAT FP111={TOOL_NO 2,BASE_NO 9,IPO_FRAME #BASE,POINT2[] " ",TQ_STATE FALSE}
DECL E6POS XP111={X -50.000,Y 40.110,Z -53.550,A 0.000,B 0.000,C -17.000}
DECL LDAT LCPDATP112={VEL 0.135,ACC 100,APO_DIST 5,APO_FAC 50.0,ORI_TYP #VAR,CIRC_TYP #BASE,JERK_FAC 50.0}
DECL FDAT FP112={TOOL_NO 2,BASE_NO 9,IPO_FRAME #BASE,POINT2[] " ",TQ_STATE FALSE}
DECL E6POS XP112={X -0.000,Y 40.110,Z -53.550,A 0.000,B 0.000,C -17.000}
DECL LDAT LCPDATP113={VEL 0.135,ACC 100,APO_DIST 5,APO_FAC 50.0,ORI_TYP #VAR,CIRC_TYP #BASE,JERK_FAC 50.0}
DECL FDAT FP113={TOOL_NO 2,BASE_NO 9,IPO_FRAME #BASE,POINT2[] " ",TQ_STATE FALSE}
DECL E6POS XP113={X 50.000,Y 40.110,Z -53.550,A 0.000,B 0.000,C -17.000}
DECL LDAT LCPDATP114={VEL 0.119,ACC 100,APO_DIST 5,APO_FAC 50.0,ORI_TYP #VAR,CIRC_TYP #BASE,JERK_FAC 50.0}
DECL FDAT FP114={TOOL_NO 2,BASE_NO 9,IPO_FRAME #BASE,POINT2[] " ",TQ_STATE FALSE}
DECL E6POS XP114={X 50.000,Y 24.230,Z -59.840,A 0.000,B 0.000,C -39.000}
DECL LDAT LCPDATP115={VEL 0.119,ACC 100,APO_DIST 5,APO_FAC 50.0,ORI_TYP #VAR,CIRC_TYP #BASE,JERK_FAC 50.0}
DECL FDAT FP115={TOOL_NO 2,BASE_NO 9,IPO_FRAME #BASE,POINT2[] " ",TQ_STATE FALSE}
DECL E6POS XP115={X -0.000,Y 24.230,Z -59.840,A 0.000,B 0.000,C -39.000}
DECL LDAT LCPDATP116={VEL 0.119,ACC 100,APO_DIST 5,APO_FAC 50.0,ORI_TYP #VAR,CIRC_TYP #BASE,JERK_FAC 50.0}
DECL FDAT FP116={TOOL_NO 2,BASE_NO 9,IPO_FRAME #BASE,POINT2[] " ",TQ_STATE FALSE}
DECL E6POS XP116={X -50.000,Y 24.230,Z -59.840,A 0.000,B 0.000,C -39.000}
DECL LDAT LCPDATP117={VEL 0.119,ACC 100,APO_DIST 5,APO_FAC 50.0,ORI_TYP #VAR,CIRC_TYP #BASE,JERK_FAC 50.0}
DECL FDAT FP117={TOOL_NO 2,BASE_NO 9,IPO_FRAME #BASE,POINT2[] " ",TQ_STATE FALSE}
DECL E6POS XP117={X -100.000,Y 24.230,Z -59.840,A 0.000,B 0.000,C -39.000}
DECL LDAT LCPDATP118={VEL 0.069,ACC 100,APO_DIST 5,APO_FAC 50.0,ORI_TYP #VAR,CIRC_TYP #BASE,JERK_FAC 50.0}
DECL FDAT FP118={TOOL_NO 2,BASE_NO 9,IPO_FRAME #BASE,POINT2[] " ",TQ_STATE FALSE}
DECL E6POS XP118={X -100.000,Y 48.790,Z -52.590,A 0.000,B 0.000,C -36.000}
DECL LDAT LCPDATP119={VEL 0.069,ACC 100,APO_DIST 5,APO_FAC 50.0,ORI_TYP #VAR,CIRC_TYP #BASE,JERK_FAC 50.0}
DECL FDAT FP119={TOOL_NO 2,BASE_NO 9,IPO_FRAME #BASE,POINT2[] " ",TQ_STATE FALSE}
DECL E6POS XP119={X -50.000,Y 48.790,Z -52.590,A 0.000,B 0.000,C -36.000}
DECL LDAT LCPDATP120={VEL 0.069,ACC 100,APO_DIST 5,APO_FAC 50.0,ORI_TYP #VAR,CIRC_TYP #BASE,JERK_FAC 50.0}
DECL FDAT FP120={TOOL_NO 2,BASE_NO 9,IPO_FRAME #BASE,POINT2[] " ",TQ_STATE FALSE}
DECL E6POS XP120={X -0.000,Y 48.790,Z -52.590,A 0.000,B 0.000,C -36.000}
DECL LDAT LCPDATP121={VEL 0.069,ACC 100,APO_DIST 5,APO_FAC 50.0,ORI_TYP #VAR,CIRC_TYP #BASE,JERK_FAC 50.0}
DECL FDAT FP121={TOOL_NO 2,BASE_NO 9,IPO_FRAME #BASE,POINT2[] " ",TQ_STATE FALSE}
DECL E6POS XP121={X 50.000,Y 48.790,Z -52.590,A 0.000,B 0.000,C -36.000}
DECL LDAT LCPDATP122={VEL 0.093,ACC 100,APO_DIST 5,APO_FAC 50.0,ORI_TYP #VAR,CIRC_TYP #BASE,JERK_FAC 50.0}
DECL FDAT FP122={TOOL_NO 2,BASE_NO 9,IPO_FRAME #BASE,POINT2[] " ",TQ_STATE FALSE}
DECL E6POS XP122={X 50.000,Y 91.140,Z -71.110,A 0.000,B 0.000,C -9.000}
DECL LDAT LCPDATP123={VEL 0.093,ACC 100,APO_DIST 5,APO_FAC 50.0,ORI_TYP #VAR,CIRC_TYP #BASE,JERK_FAC 50.0}
DECL FDAT FP123={TOOL_NO 2,BASE_NO 9,IPO_FRAME #BASE,POINT2[] " ",TQ_STATE FALSE}
DECL E6POS XP123={X -0.000,Y 91.140,Z -71.110,A 0.000,B 0.000,C -9.000}
DECL LDAT LCPDATP124={VEL 0.093,ACC 100,APO_DIST 5,APO_FAC 50.0,ORI_TYP #VAR,CIRC_TYP #BASE,JERK_FAC 50.0}
DECL FDAT FP124={TOOL_NO 2,BASE_NO 9,IPO_FRAME #BASE,POINT2[] " ",TQ_STATE FALSE}
DECL E6POS XP124={X -50.000,Y 91.140,Z -71.110,A 0.000,B 0.000,C -9.000}
DECL LDAT LCPDATP125={VEL 0.093,ACC 100,APO_DIST 5,APO_FAC 50.0,ORI_TYP #VAR,CIRC_TYP #BASE,JERK_FAC 50.0}
DECL FDAT FP125={TOOL_NO 2,BASE_NO 9,IPO_FRAME #BASE,POINT2[] " ",TQ_STATE FALSE}
DECL E6POS XP125={X -100.000,Y 91.140,Z -71.110,A 0.000,B 0.000,C -9.000}
DECL LDAT LCPDATP126={VEL 0.072,ACC 100,APO_DIST 5,APO_FAC 50.0,ORI_TYP #VAR,CIRC_TYP #BASE,JERK_FAC 50.0}
DECL FDAT FP126={TOOL_NO 2,BASE_NO 9,IPO_FRAME #BASE,POINT2[] " ",TQ_STATE FALSE}
DECL E6POS XP126={X -100.000,Y 100.110,Z -53.550,A 0.000,B 0.000,C -17.000}
DECL LDAT LCPDATP127={VEL 0.072,ACC 100,APO_DIST 5,APO_FAC 50.0,ORI_TYP #VAR,CIRC_TYP #BASE,JERK_FAC 50.0}
DECL FDAT FP127={TOOL_NO 2,BASE_NO 9,IPO_FRAME #BASE,POINT2[] " ",TQ_STATE FALSE}
DECL E6POS XP127={X -50.000,Y 100.110,Z -53.550,A 0.000,B 0.000,C -17.000}
DECL LDAT LCPDATP128={VEL 0.072,ACC 100,APO_DIST 5,APO_FAC 50.0,ORI_TYP #VAR,CIRC_TYP #BASE,JERK_FAC 50.0}
DECL FDAT FP128={TOOL_NO 2,BASE_NO 9,IPO_FRAME #BASE,POINT2[] " ",TQ_STATE FALSE}
DECL E6POS XP128={X -0.000,Y 100.110,Z -53.550,A 0.000,B 0.000,C -17.000}
DECL LDAT LCPDATP129={VEL 0.072,ACC 100,APO_DIST 5,APO_FAC 50.0,ORI_TYP #VAR,CIRC_TYP #BASE,JERK_FAC 50.0}
DECL FDAT FP129={TOOL_NO 2,BASE_NO 9,IPO_FRAME #BASE,POINT2[] " ",TQ_STATE FALSE}
DECL E6POS XP129={X 50.000,Y 100.110,Z -53.550,A 0.000,B 0.000,C -17.000}
DECL LDAT LCPDATP130={VEL 0.148,ACC 100,APO_DIST 5,APO_FAC 50.0,ORI_TYP #VAR,CIRC_TYP #BASE,JERK_FAC 50.0}
DECL FDAT FP130={TOOL_NO 2,BASE_NO 9,IPO_FRAME #BASE,POINT2[] " ",TQ_STATE FALSE}
DECL E6POS XP130={X 50.000,Y 97.570,Z -52.840,A 0.000,B 0.000,C -33.000}
DECL LDAT LCPDATP131={VEL 0.148,ACC 100,APO_DIST 5,APO_FAC 50.0,ORI_TYP #VAR,CIRC_TYP #BASE,JERK_FAC 50.0}
DECL FDAT FP131={TOOL_NO 2,BASE_NO 9,IPO_FRAME #BASE,POINT2[] " ",TQ_STATE FALSE}
DECL E6POS XP131={X -0.000,Y 97.570,Z -52.840,A 0.000,B 0.000,C -33.000}
DECL LDAT LCPDATP132={VEL 0.148,ACC 100,APO_DIST 5,APO_FAC 50.0,ORI_TYP #VAR,CIRC_TYP #BASE,JERK_FAC 50.0}
DECL FDAT FP132={TOOL_NO 2,BASE_NO 9,IPO_FRAME #BASE,POINT2[] " ",TQ_STATE FALSE}
DECL E6POS XP132={X -50.000,Y 97.570,Z -52.840,A 0.000,B 0.000,C -33.000}
DECL LDAT LCPDATP133={VEL 0.148,ACC 100,APO_DIST 5,APO_FAC 50.0,ORI_TYP #VAR,CIRC_TYP #BASE,JERK_FAC 50.0}
DECL FDAT FP133={TOOL_NO 2,BASE_NO 9,IPO_FRAME #BASE,POINT2[] " ",TQ_STATE FALSE}
DECL E6POS XP133={X -100.000,Y 97.570,Z -52.840,A 0.000,B 0.000,C -33.000}
DECL LDAT LCPDATP134={VEL 0.055,ACC 100,APO_DIST 5,APO_FAC 50.0,ORI_TYP #VAR,CIRC_TYP #BASE,JERK_FAC 50.0}
DECL FDAT FP134={TOOL_NO 2,BASE_NO 9,IPO_FRAME #BASE,POINT2[] " ",TQ_STATE FALSE}
DECL E6POS XP134={X -100.000,Y 134.600,Z -45.600,A 0.000,B 0.000,C -14.000}
DECL LDAT LCPDATP135={VEL 0.055,ACC 100,APO_DIST 5,APO_FAC 50.0,ORI_TYP #VAR,CIRC_TYP #BASE,JERK_FAC 50.0}
DECL FDAT FP135={TOOL_NO 2,BASE_NO 9,IPO_FRAME #BASE,POINT2[] " ",TQ_STATE FALSE}
DECL E6POS XP135={X -50.000,Y 134.600,Z -45.600,A 0.000,B 0.000,C -14.000}
DECL LDAT LCPDATP136={VEL 0.055,ACC 100,APO_DIST 5,APO_FAC 50.0,ORI_TYP #VAR,CIRC_TYP #BASE,JERK_FAC 50.0}
DECL FDAT FP136={TOOL_NO 2,BASE_NO 9,IPO_FRAME #BASE,POINT2[] " ",TQ_STATE FALSE}
DECL E6POS XP136={X -0.000,Y 134.600,Z -45.600,A 0.000,B 0.000,C -14.000}
DECL LDAT LCPDATP137={VEL 0.055,ACC 100,APO_DIST 5,APO_FAC 50.0,ORI_TYP #VAR,CIRC_TYP #BASE,JERK_FAC 50.0}
DECL FDAT FP137={TOOL_NO 2,BASE_NO 9,IPO_FRAME #BASE,POINT2[] " ",TQ_STATE FALSE}
DECL E6POS XP137={X 50.000,Y 134.600,Z -45.600,A 0.000,B 0.000,C -14.000}
DECL LDAT LCPDATP138={VEL 0.149,ACC 100,APO_DIST 5,APO_FAC 50.0,ORI_TYP #VAR,CIRC_TYP #BASE,JERK_FAC 50.0}
DECL FDAT FP138={TOOL_NO 2,BASE_NO 9,IPO_FRAME #BASE,POINT2[] " ",TQ_STATE FALSE}
DECL E6POS XP138={X 50.000,Y 142.850,Z -89.640,A 0.000,B 0.000,C -13.000}
DECL LDAT LCPDATP139={VEL 0.149,ACC 100,APO_DIST 5,APO_FAC 50.0,ORI_TYP #VAR,CIRC_TYP #BASE,JERK_FAC 50.0}
DECL FDAT FP139={TOOL_NO 2,BASE_NO 9,IPO_FRAME #BASE,POINT2[] " ",TQ_STATE FALSE}
DECL E6POS XP139={X -0.000,Y 142.850,Z -89.640,A 0.000,B 0.000,C -13.000}
DECL LDAT LCPDATP140={VEL 0.149,ACC 100,APO_DIST 5,APO_FAC 50.0,ORI_TYP #VAR,CIRC_TYP #BASE,JERK_FAC 50.0}
DECL FDAT FP140={TOOL_NO 2,BASE_NO 9,IPO_FRAME #BASE,POINT2[] " ",TQ_STATE FALSE}
DECL E6POS XP140={X -50.000,Y 142.850,Z -89.640,A 0.000,B 0.000,C -13.000}
DECL LDAT LCPDATP141={VEL 0.149,ACC 100,APO_DIST 5,APO_FAC 50.0,ORI_TYP #VAR,CIRC_TYP #BASE,JERK_FAC 50.0}
DECL FDAT FP141={TOOL_NO 2,BASE_NO 9,IPO_FRAME #BASE,POINT2[] " ",TQ_STATE FALSE}
DECL E6POS XP141={X -100.000,Y 142.850,Z -89.640,A 0.000,B 0.000,C -13.000}
DECL LDAT LCPDATP142={VEL 0.101,ACC 100,APO_DIST 5,APO_FAC 50.0,ORI_TYP #VAR,CIRC_TYP #BASE,JERK_FAC 50.0}
DECL FDAT FP142={TOOL_NO 2,BASE_NO 9,IPO_FRAME #BASE,POINT2[] " ",TQ_STATE FALSE}
DECL E6POS XP142={X -100.000,Y 141.950,Z -67.100,A 0.000,B 0.000,C -28.000}
DECL LDAT LCPDATP143={VEL 0.101,ACC 100,APO_DIST 5,APO_FAC 50.0,ORI_TYP #VAR,CIRC_TYP #BASE,JERK_FAC 50.0}
DECL FDAT FP143={TOOL_NO 2,BASE_NO 9,IPO_FRAME #BASE,POINT2[] " ",TQ_STATE FALSE}
DECL E6POS XP143={X -50.000,Y 141.950,Z -67.100,A 0.000,B 0.000,C -28.000}
DECL LDAT LCPDATP144={VEL 0.101,ACC 100,APO_DIST 5,APO_FAC 50.0,ORI_TYP #VAR,CIRC_TYP #BASE,JERK_FAC 50.0}
DECL FDAT FP144={TOOL_NO 2,BASE_NO 9,IPO_FRAME #BASE,POINT2[] " ",TQ_STATE FALSE}
DECL E6POS XP144={X -0.000,Y 141.950,Z -67.100,A 0.000,B 0.000,C -28.000}
DECL LDAT LCPDATP145={VEL 0.101,ACC 100,APO_DIST 5,APO_FAC 50.0,ORI_TYP #VAR,CIRC_TYP #BASE,JERK_FAC 50.0}
DECL FDAT FP145={TOOL_NO 2,BASE_NO 9,IPO_FRAME #BASE,POINT2[] " ",TQ_STATE FALSE}
DECL E6POS XP145={X 50.000,Y 141.950,Z -67.100,A 0.000,B 0.000,C -28.000}
DECL LDAT LCPDATP146={VEL 0.071,ACC 100,APO_DIST 5,APO_FAC 50.0,ORI_TYP #VAR,CIRC_TYP #BASE,JERK_FAC 50.0}
DECL FDAT FP146={TOOL_NO 2,BASE_NO 9,IPO_FRAME #BASE,POINT2[] " ",TQ_STATE FALSE}
DECL E6POS XP146={X 50.000,Y 189.020,Z -32.980,A 0.000,B 0.000,C -2.000}
DECL LDAT LCPDATP147={VEL 0.071,ACC 100,APO_DIST 5,APO_FAC 50.0,ORI_TYP #VAR,CIRC_TYP #BASE,JERK_FAC 50.0}
DECL FDAT FP147={TOOL_NO 2,BASE_NO 9,IPO_FRAME #BASE,POINT2[] " ",TQ_STATE FALSE}
DECL E6POS XP147={X -0.000,Y 189.020,Z -32.980,A 0.000,B 0.000,C -2.000}
DECL LDAT LCPDATP148={VEL 0.071,ACC 100,APO_DIST 5,APO_FAC 50.0,ORI_TYP #VAR,CIRC_TYP #BASE,JERK_FAC 50.0}
DECL FDAT FP148={TOOL_NO 2,BASE_NO 9,IPO_FRAME #BASE,POINT2[] " ",TQ_STATE FALSE}
DECL E6POS XP148={X -50.000,Y 189.020,Z -32.980,A 0.000,B 0.000,C -2.000}
DECL LDAT LCPDATP149={VEL 0.071,ACC 100,APO_DIST 5,APO_FAC 50.0,ORI_TYP #VAR,CIRC_TYP #BASE,JERK_FAC 50.0}
DECL FDAT FP149={TOOL_NO 2,BASE_NO 9,IPO_FRAME #BASE,POINT2[] " ",TQ_STATE FALSE}
DECL E6POS XP149={X -100.000,Y 189.020,Z -32.980,A 0.000,B 0.000,C -2.000}
DECL LDAT LCPDATP150={VEL 0.121,ACC 100,APO_DIST 5,APO_FAC 50.0,ORI_TYP #VAR,CIRC_TYP #BASE,JERK_FAC 50.0}
DECL FDAT FP150={TOOL_NO 2,BASE_NO 9,IPO_FRAME #BASE,POINT2[] " ",TQ_STATE FALSE}
DECL E6POS XP150={X -100.000,Y 199.670,Z -30.530,A 0.000,B 0.000,C -10.000}
DECL LDAT LCPDATP151={VEL 0.121,ACC 100,APO_DIST 5,APO_FAC 50.0,ORI_TYP #VAR,CIRC_TYP #BASE,JERK_FAC 50.0}
DECL FDAT FP151={TOOL_NO 2,BASE_NO 9,IPO_FRAME #BASE,POINT2[] " ",TQ_STATE FALSE}
DECL E6POS XP151={X -50.000,Y 199.670,Z -30.530,A 0.000,B 0.000,C -10.000}
DECL LDAT LCPDATP152={VEL 0.121,ACC 100,APO_DIST 5,APO_FAC 50.0,ORI_TYP #VAR,CIRC_TYP #BASE,JERK_FAC 50.0}
DECL FDAT FP152={TOOL_NO 2,BASE_NO 9,IPO_FRAME #BASE,POINT2[] " ",TQ_STATE FALSE}
DECL E6POS XP152={X -0.000,Y 199.670,Z -30.530,A 0.000,B 0.000,C -10.000}
DECL LDAT LCPDATP153={VEL 0.121,ACC 100,APO_DIST 5,APO_FAC 50.0,ORI_TYP #VAR,CIRC_TYP #BASE,JERK_FAC 50.0}
DECL FDAT FP153={TOOL_NO 2,BASE_NO 9,IPO_FRAME #BASE,POINT2[] " ",TQ_STATE FALSE}
DECL E6POS XP153={X 50.000,Y 199.670,Z -30.530,A 0.000,B 0.000,C -10.000}
DECL LDAT LCPDATP154={VEL 0.061,ACC 100,APO_DIST 5,APO_FAC 50.0,ORI_TYP #VAR,CIRC_TYP #BASE,JERK_FAC 50.0}
DECL FDAT FP154={TOOL_NO 2,BASE_NO 9,IPO_FRAME #BASE,POINT2[] " ",TQ_STATE FALSE}
DECL E6POS XP154={X 50.000,Y 202.790,Z -30.310,A 0.000,B 0.000,C -30.000}
DECL LDAT LCPDATP155={VEL 0.061,ACC 100,APO_DIST 5,APO_FAC 50.0,ORI_TYP #VAR,CIRC_TYP #BASE,JERK_FAC 50.0}
DECL FDAT FP155={TOOL_NO 2,BASE_NO 9,IPO_FRAME #BASE,POINT2[] " ",TQ_STATE FALSE}
DECL E6POS XP155={X -0.000,Y 202.790,Z -30.310,A 0.000,B 0.000,C -30.000}
DECL LDAT LCPDATP156={VEL 0.061,ACC 100,APO_DIST 5,APO_FAC 50.0,ORI_TYP #VAR,CIRC_TYP #BASE,JERK_FAC 50.0}
DECL FDAT FP156={TOOL_NO 2,BASE_NO 9,IPO_FRAME #BASE,POINT2[] " ",TQ_STATE FALSE}
DECL E6POS XP156={X -50.000,Y 202.790,Z -30.310,A 0.000,B 0.000,C -30.000}
DECL LDAT LCPDATP157={VEL 0.061,ACC 100,APO_DIST 5,APO_FAC 50.0,ORI_TYP #VAR,CIRC_TYP #BASE,JERK_FAC 50.0}
DECL FDAT FP157={TOOL_NO 2,BASE_NO 9,IPO_FRAME #BASE,POINT2[] " ",TQ_STATE FALSE}
DECL E6POS XP157={X -100.000,Y 202.790,Z -30.310,A 0.000,B 0.000,C -30.000}
DECL LDAT LCPDATP158={VEL 0.5,ACC 100,APO_DIST 5,APO_FAC 50.0,ORI_TYP #VAR,CIRC_TYP #BASE,JERK_FAC 50.0}
DECL FDAT FP158={TOOL_NO 2,BASE_NO 9,IPO_FRAME #BASE,POINT2[] " ",TQ_STATE FALSE}
DECL E6POS XP158={X -150.000,Y 220.290,Z -50.000,A 0.000,B 0.000,C 0.000}
DECL LDAT LCPDATP159={VEL 1.0,ACC 100,APO_DIST 5,APO_FAC 50.0,ORI_TYP #VAR,CIRC_TYP #BASE,JERK_FAC 50.0}
DECL FDAT FP159={TOOL_NO 2,BASE_NO 9,IPO_FRAME #BASE,POINT2[] " ",TQ_STATE FALSE}
DECL E6POS XP159={X -150.000,Y 260.000,Z -20.000,A 0.000,B 0.000,C 0.000}
DECL LDAT LCPDATP160={VEL 1.0,ACC 100,APO_DIST 5,APO_FAC 50.0,ORI_TYP #VAR,CIRC_TYP #BASE,JERK_FAC 50.0}
DECL FDAT FP160={TOOL_NO 2,BASE_NO 9,IPO_FRAME #BASE,POINT2[] " ",TQ_STATE FALSE}
DECL E6POS XP160={X 100.000,Y 260.000,Z -20.000,A 0.000,B 0.000,C 0.000}
;ENDDAT for Routine_1


; Data for Routine_2
DECL LDAT LCPDATP161={VEL 1.0,ACC 100,APO_DIST 5,APO_FAC 50.0,ORI_TYP #VAR,CIRC_TYP #BASE,JERK_FAC 50.0}
DECL FDAT FP161={TOOL_NO 2,BASE_NO 8,IPO_FRAME #BASE,POINT2[] " ",TQ_STATE FALSE}
DECL E6POS XP161={X 100.000,Y 0.000,Z -100.000,A 0.000,B 0.000,C 0.000}
DECL LDAT LCPDATP162={VEL 0.123,ACC 100,APO_DIST 5,APO_FAC 50.0,ORI_TYP #VAR,CIRC_TYP #BASE,JERK_FAC 50.0}
DECL FDAT FP162={TOOL_NO 2,BASE_NO 8,IPO_FRAME #BASE,POINT2[] " ",TQ_STATE FALSE}
DECL E6POS XP162={X 50.000,Y -12.510,Z -68.600,A 0.000,B 0.000,C -20.000}
DECL LDAT LCPDATP163={VEL 0.123,ACC 100,APO_DIST 5,APO_FAC 50.0,ORI_TYP #VAR,CIRC_TYP #BASE,JERK_FAC 50.0}
DECL FDAT FP163={TOOL_NO 2,BASE_NO 8,IPO_FRAME #BASE,POINT2[] " ",TQ_STATE FALSE}
DECL E6POS XP163={X 0.000,Y -12.510,Z -68.600,A 0.000,B 0.000,C -20.000}
DECL LDAT LCPDATP164={VEL 0.123,ACC 100,APO_DIST 5,APO_FAC 50.0,ORI_TYP #VAR,CIRC_TYP #BASE,JERK_FAC 50.0}
DECL FDAT FP164={TOOL_NO 2,BASE_NO 8,IPO_FRAME #BASE,POINT2[] " ",TQ_STATE FALSE}
DECL E6POS XP164={X -50.000,Y -12.510,Z -68.600,A 0.000,B 0.000,C -20.000}
DECL LDAT LCPDATP165={VEL 0.123,ACC 100,APO_DIST 5,APO_FAC 50.0,ORI_TYP #VAR,CIRC_TYP #BASE,JERK_FAC 50.0}
DECL FDAT FP165={TOOL_NO 2,BASE_NO 8,IPO_FRAME #BASE,POINT2[] " ",TQ_STATE FALSE}
DECL E6POS XP165={X -100.000,Y -12.510,Z -68.600,A 0.000,B 0.000,C -20.000}
DECL LDAT LCPDATP166={VEL 0.128,ACC 100,APO_DIST 5,APO_FAC 50.0,ORI_TYP #VAR,CIRC_TYP #BASE,JERK_FAC 50.0}
DECL FDAT FP166={TOOL_NO 2,BASE_NO 8,IPO_FRAME #BASE,POINT2[] " ",TQ_STATE FALSE}
DECL E6POS XP166={X -100.000,Y -8.150,Z -77.940,A 0.000,B 0.000,C -25.000}
DECL LDAT LCPDATP167={VEL 0.128,ACC 100,APO_DIST 5,APO_FAC 50.0,ORI_TYP #VAR,CIRC_TYP #BASE,JERK_FAC 50.0}
DECL FDAT FP167={TOOL_NO 2,BASE_NO 8,IPO_FRAME #BASE,POINT2[] " ",TQ_STATE FALSE}
DECL E6POS XP167={X -50.000,Y -8.150,Z -77.940,A 0.000,B 0.000,C -25.000}
DECL LDAT LCPDATP168={VEL 0.128,ACC 100,APO_DIST 5,APO_FAC 50.0,ORI_TYP #VAR,CIRC_TYP #BASE,JERK_FAC 50.0}
DECL FDAT FP168={TOOL_NO 2,BASE_NO 8,IPO_FRAME #BASE,POINT2[] " ",TQ_STATE FALSE}
DECL E6POS XP168={X 0.000,Y -8.150,Z -77.940,A 0.000,B 0.000,C -25.000}
DECL LDAT LCPDATP169={VEL 0.128,ACC 100,APO_DIST 5,APO_FAC 50.0,ORI_TYP #VAR,CIRC_TYP #BASE,JERK_FAC 50.0}
DECL FDAT FP169={TOOL_NO 2,BASE_NO 8,IPO_FRAME #BASE,POINT2[] " ",TQ_STATE FALSE}
DECL E6POS XP169={X 50.000,Y -8.150,Z -77.940,A 0.000,B 0.000,C -25.000}
DECL LDAT LCPDATP170={VEL 0.103,ACC 100,APO_DIST 5,APO_FAC 50.0,ORI_TYP #VAR,CIRC_TYP #BASE,JERK_FAC 50.0}
DECL FDAT FP170={TOOL_NO 2,BASE_NO 8,IPO_FRAME #BASE,POINT2[] " ",TQ_STATE FALSE}
DECL E6POS XP170={X 50.000,Y 41.710,Z -60.000,A 0.000,B 0.000,C 0.000}
DECL LDAT LCPDATP171={VEL 0.103,ACC 100,APO_DIST 5,APO_FAC 50.0,ORI_TYP #VAR,CIRC_TYP #BASE,JERK_FAC 50.0}
DECL FDAT FP171={TOOL_NO 2,BASE_NO 8,IPO_FRAME #BASE,POINT2[] " ",TQ_STATE FALSE}
DECL E6POS XP171={X -0.000,Y 41.710,Z -60.000,A 0.000,B 0.000,C 0.000}
DECL LDAT LCPDATP172={VEL 0.103,ACC 100,APO_DIST 5,APO_FAC 50.0,ORI_TYP #VAR,CIRC_TYP #BASE,JERK_FAC 50.0}
DECL FDAT FP172={TOOL_NO 2,BASE_NO 8,IPO_FRAME #BASE,POINT2[] " ",TQ_STATE FALSE}
DECL E6POS XP172={X -50.000,Y 41.710,Z -60.000,A 0.000,B 0.000,C 0.000}
DECL LDAT LCPDATP173={VEL 0.103,ACC 100,APO_DIST 5,APO_FAC 50.0,ORI_TYP #VAR,CIRC_TYP #BASE,JERK_FAC 50.0}
DECL FDAT FP173={TOOL_NO 2,BASE_NO 8,IPO_FRAME #BASE,POINT2[] " ",TQ_STATE FALSE}
DECL E6POS XP173={X -100.000,Y 41.710,Z -60.000,A 0.000,B 0.000,C 0.000}
DECL LDAT LCPDATP174={VEL 0.108,ACC 100,APO_DIST 5,APO_FAC 50.0,ORI_TYP #VAR,CIRC_TYP #BASE,JERK_FAC 50.0}
DECL FDAT FP174={TOOL_NO 2,BASE_NO 8,IPO_FRAME #BASE,POINT2[] " ",TQ_STATE FALSE}
DECL E6POS XP174={X -100.000,Y 43.810,Z -45.400,A 0.000,B 0.000,C -15.000}
DECL LDAT LCPDATP175={VEL 0.108,ACC 100,APO_DIST 5,APO_FAC 50.0,ORI_TYP #VAR,CIRC_TYP #BASE,JERK_FAC 50.0}
DECL FDAT FP175={TOOL_NO 2,BASE_NO 8,IPO_FRAME #BASE,POINT2[] " ",TQ_STATE FALSE}
DECL E6POS XP175={X -50.000,Y 43.810,Z -45.400,A 0.000,B 0.000,C -15.000}
DECL LDAT LCPDATP176={VEL 0.108,ACC 100,APO_DIST 5,APO_FAC 50.0,ORI_TYP #VAR,CIRC_TYP #BASE,JERK_FAC 50.0}
DECL FDAT FP176={TOOL_NO 2,BASE_NO 8,IPO_FRAME #BASE,POINT2[] " ",TQ_STATE FALSE}
DECL E6POS XP176={X -0.000,Y 43.810,Z -45.400,A 0.000,B 0.000,C -15.000}
DECL LDAT LCPDATP177={VEL 0.108,ACC 100,APO_DIST 5,APO_FAC 50.0,ORI_TYP #VAR,CIRC_TYP #BASE,JERK_FAC 50.0}
DECL FDAT FP177={TOOL_NO 2,BASE_NO 8,IPO_FRAME #BASE,POINT2[] " ",TQ_STATE FALSE}
DECL E6POS XP177={X 50.000,Y 43.810,Z -45.400,A 0.000,B 0.000,C -15.000}
DECL LDAT LCPDATP178={VEL 0.095,ACC 100,APO_DIST 5,APO_FAC 50.0,ORI_TYP #VAR,CIRC_TYP #BASE,JERK_FAC 50.0}
DECL FDAT FP178={TOOL_NO 2,BASE_NO 8,IPO_FRAME #BASE,POINT2[] " ",TQ_STATE FALSE}
DECL E6POS XP178={X 50.000,Y 50.270,Z -49.710,A 0.000,B 0.000,C -23.000}
DECL LDAT LCPDATP179={VEL 0.095,ACC 100,APO_DIST 5,APO_FAC 50.0,ORI_TYP #VAR,CIRC_TYP #BASE,JERK_FAC 50.0}
DECL FDAT FP179={TOOL_NO 2,BASE_NO 8,IPO_FRAME #BASE,POINT2[] " ",TQ_STATE FALSE}
DECL E6POS XP179={X -0.000,Y 50.270,Z -49.710,A 0.000,B 0.000,C -23.000}
DECL LDAT LCPDATP180={VEL 0.095,ACC 100,APO_DIST 5,APO_FAC 50.0,ORI_TYP #VAR,CIRC_TYP #BASE,JERK_FAC 50.0}
DECL FDAT FP180={TOOL_NO 2,BASE_NO 8,IPO_FRAME #BASE,POINT2[] " ",TQ_STATE FALSE}
DECL E6POS XP180={X -50.000,Y 50.270,Z -49.710,A 0.000,B 0.000,C -23.000}
DECL LDAT LCPDATP181={VEL 0.095,ACC 100,APO_DIST 5,APO_FAC 50.0,ORI_TYP #VAR,CIRC_TYP #BASE,JERK_FAC 50.0}
DECL FDAT FP181={TOOL_NO 2,BASE_NO 8,IPO_FRAME #BASE,POINT2[] " ",TQ_STATE FALSE}
DECL E6POS XP181={X -100.000,Y 50.270,Z -49.710,A 0.000,B 0.000,C -23.000}
DECL LDAT LCPDATP182={VEL 0.142,ACC 100,APO_DIST 5,APO_FAC 50.0,ORI_TYP #VAR,CIRC_TYP #BASE,JERK_FAC 50.0}
DECL FDAT FP182={TOOL_NO 2,BASE_NO 8,IPO_FRAME #BASE,POINT2[] " ",TQ_STATE FALSE}
DECL E6POS XP182={X -100.000,Y 77.240,Z -35.080,A 0.000,B 0.000,C -13.000}
DECL LDAT LCPDATP183={VEL 0.142,ACC 100,APO_DIST 5,APO_FAC 50.0,ORI_TYP #VAR,CIRC_TYP #BASE,JERK_FAC 50.0}
DECL FDAT FP183={TOOL_NO 2,BASE_NO 8,IPO_FRAME #BASE,POINT2[] " ",TQ_STATE FALSE}
DECL E6POS XP183={X -50.000,Y 77.240,Z -35.080,A 0.000,B 0.000,C -13.000}
DECL LDAT LCPDATP184={VEL 0.142,ACC 100,APO_DIST 5,APO_FAC 50.0,ORI_TYP #VAR,CIRC_TYP #BASE,JERK_FAC 50.0}
DECL FDAT FP184={TOOL_NO 2,BASE_NO 8,IPO_FRAME #BASE,POINT2[] " ",TQ_STATE FALSE}
DECL E6POS XP184={X -0.000,Y 77.240,Z -35.080,A 0.000,B 0.000,C -13.000}
DECL LDAT LCPDATP185={VEL 0.142,ACC 100,APO_DIST 5,APO_FAC 50.0,ORI_TYP #VAR,CIRC_TYP #BASE,JERK_FAC 50.0}
DECL FDAT FP185={TOOL_NO 2,BASE_NO 8,IPO_FRAME #BASE,POINT2[] " ",TQ_STATE FALSE}
DECL E6POS XP185={X 50.000,Y 77.240,Z -35.080,A 0.000,B 0.000,C -13.000}
DECL LDAT LCPDATP186={VEL 0.142,ACC 100,APO_DIST 5,APO_FAC 50.0,ORI_TYP #VAR,CIRC_TYP #BASE,JERK_FAC 50.0}
DECL FDAT FP186={TOOL_NO 2,BASE_NO 8,IPO_FRAME #BASE,POINT2[] " ",TQ_STATE FALSE}
DECL E6POS XP186={X 50.000,Y 94.780,Z -73.590,A 0.000,B 0.000,C -6.000}
DECL LDAT LCPDATP187={VEL 0.142,ACC 100,APO_DIST 5,APO_FAC 50.0,ORI_TYP #VAR,CIRC_TYP #BASE,JERK_FAC 50.0}
DECL FDAT FP187={TOOL_NO 2,BASE_NO 8,IPO_FRAME #BASE,POINT2[] " ",TQ_STATE FALSE}
DECL E6POS XP187={X -0.000,Y 94.780,Z -73.590,A 0.000,B 0.000,C -6.000}
DECL LDAT LCPDATP188={VEL 0.142,ACC 100,APO_DIST 5,APO_FAC 50.0,ORI_TYP #VAR,CIRC_TYP #BASE,JERK_FAC 50.0}
DECL FDAT FP188={TOOL_NO 2,BASE_NO 8,IPO_FRAME #BASE,POINT2[] " ",TQ_STATE FALSE}
DECL E6POS XP188={X -50.000,Y 94.780,Z -73.590,A 0.000,B 0.000,C -6.000}
DECL LDAT LCPDATP189={VEL 0.142,ACC 100,APO_DIST 5,APO_FAC 50.0,ORI_TYP #VAR,CIRC_TYP #BASE,JERK_FAC 50.0}
DECL FDAT FP189={TOOL_NO 2,BASE_NO 8,IPO_FRAME #BASE,POINT2[] " ",TQ_STATE FALSE}
DECL E6POS XP189={X -100.000,Y 94.780,Z -73.590,A 0.000,B 0.000,C -6.000}
DECL LDAT LCPDATP190={VEL 0.064,ACC 100,APO_DIST 5,APO_FAC 50.0,ORI_TYP #VAR,CIRC_TYP #BASE,JERK_FAC 50.0}
DECL FDAT FP190={TOOL_NO 2,BASE_NO 8,IPO_FRAME #BASE,POINT2[] " ",TQ_STATE FALSE}
DECL E6POS XP190={X -100.000,Y 84.800,Z -40.190,A 0.000,B 0.000,C -38.000}
DECL LDAT LCPDATP191={VEL 0.064,ACC 100,APO_DIST 5,APO_FAC 50.0,ORI_TYP #VAR,CIRC_TYP #BASE,JERK_FAC 50.0}
DECL FDAT FP191={TOOL_NO 2,BASE_NO 8,IPO_FRAME #BASE,POINT2[] " ",TQ_STATE FALSE}
DECL E6POS XP191={X -50.000,Y 84.800,Z -40.190,A 0.000,B 0.000,C -38.000}
DECL LDAT LCPDATP192={VEL 0.064,ACC 100,APO_DIST 5,APO_FAC 50.0,ORI_TYP #VAR,CIRC_TYP #BASE,JERK_FAC 50.0}
DECL FDAT FP192={TOOL_NO 2,BASE_NO 8,IPO_FRAME #BASE,POINT2[] " ",TQ_STATE FALSE}
DECL E6POS XP192={X -0.000,Y 84.800,Z -40.190,A 0.000,B 0.000,C -38.000}
DECL LDAT LCPDATP193={VEL 0.064,ACC 100,APO_DIST 5,APO_FAC 50.0,ORI_TYP #VAR,CIRC_TYP #BASE,JERK_FAC 50.0}
DECL FDAT FP193={TOOL_NO 2,BASE_NO 8,IPO_FRAME #BASE,POINT2[] " ",TQ_STATE FALSE}
DECL E6POS XP193={X 50.000,Y 84.800,Z -40.190,A 0.000,B 0.000,C -38.000}
DECL LDAT LCPDATP194={VEL 0.055,ACC 100,APO_DIST 5,APO_FAC 50.0,ORI_TYP #VAR,CIRC_TYP #BASE,JERK_FAC 50.0}
DECL FDAT FP194={TOOL_NO 2,BASE_NO 8,IPO_FRAME #BASE,POINT2[] " ",TQ_STATE FALSE}
DECL E6POS XP194={X 50.000,Y 76.790,Z -69.940,A 0.000,B 0.000,C -39.000}
DECL LDAT LCPDATP195={VEL 0.055,ACC 100,APO_DIST 5,APO_FAC 50.0,ORI_TYP #VAR,CIRC_TYP #BASE,JERK_FAC 50.0}
DECL FDAT FP195={TOOL_NO 2,BASE_NO 8,IPO_FRAME #BASE,POINT2[] " ",TQ_STATE FALSE}
DECL E6POS XP195={X -0.000,Y 76.790,Z -69.940,A 0.000,B 0.000,C -39.000}
DECL LDAT LCPDATP196={VEL 0.055,ACC 100,APO_DIST 5,APO_FAC 50.0,ORI_TYP #VAR,CIRC_TYP #BASE,JERK_FAC 50.0}
DECL FDAT FP196={TOOL_NO 2,BASE_NO 8,IPO_FRAME #BASE,POINT2[] " ",TQ_STATE FALSE}
DECL E6POS XP196={X -50.000,Y 76.790,Z -69.940,A 0.000,B 0.000,C -39.000}
DECL LDAT LCPDATP197={VEL 0.055,ACC 100,APO_DIST 5,APO_FAC 50.0,ORI_TYP #VAR,CIRC_TYP #BASE,JERK_FAC 50.0}
DECL FDAT FP197={TOOL_NO 2,BASE_NO 8,IPO_FRAME #BASE,POINT2[] " ",TQ_STATE FALSE}
DECL E6POS XP197={X -100.000,Y 76.790,Z -69.940,A 0.000,B 0.000,C -39.000}
DECL LDAT LCPDATP198={VEL 0.12,ACC 100,APO_DIST 5,APO_FAC 50.0,ORI_TYP #VAR,CIRC_TYP #BASE,JERK_FAC 50.0}
DECL FDAT FP198={TOOL_NO 2,BASE_NO 8,IPO_FRAME #BASE,POINT2[] " ",TQ_STATE FALSE}
DECL E6POS XP198={X -100.000,Y 132.190,Z -81.480,A 0.000,B 0.000,C -11.000}
DECL LDAT LCPDATP199={VEL 0.12,ACC 100,APO_DIST 5,APO_FAC 50.0,ORI_TYP #VAR,CIRC_TYP #BASE,JERK_FAC 50.0}
DECL FDAT FP199={TOOL_NO 2,BASE_NO 8,IPO_FRAME #BASE,POINT2[] " ",TQ_STATE FALSE}
DECL E6POS XP199={X -50.000,Y 132.190,Z -81.480,A 0.000,B 0.000,C -11.000}
DECL LDAT LCPDATP200={VEL 0.12,ACC 100,APO_DIST 5,APO_FAC 50.0,ORI_TYP #VAR,CIRC_TYP #BASE,JERK_FAC 50.0}
DECL FDAT FP200={TOOL_NO 2,BASE_NO 8,IPO_FRAME #BASE,POINT2[] " ",TQ_STATE FALSE}
DECL E6POS XP200={X -0.000,Y 132.190,Z -81.480,A 0.000,B 0.000,C -11.000}
DECL LDAT LCPDATP201={VEL 0.12,ACC 100,APO_DIST 5,APO_FAC 50.0,ORI_TYP #VAR,CIRC_TYP #BASE,JERK_FAC 50.0}
DECL FDAT FP201={TOOL_NO 2,BASE_NO 8,IPO_FRAME #BASE,POINT2[] " ",TQ_STATE FALSE}
DECL E6POS XP201={X 50.000,Y 132.190,Z -81.480,A 0.000,B 0.000,C -11.000}
DECL LDAT LCPDATP202={VEL 0.081,ACC 100,APO_DIST 5,APO_FAC 50.0,ORI_TYP #VAR,CIRC_TYP #BASE,JERK_FAC 50.0}
DECL FDAT FP202={TOOL_NO 2,BASE_NO 8,IPO_FRAME #BASE,POINT2[] " ",TQ_STATE FALSE}
DECL E6POS XP202={X 50.000,Y 124.070,Z -69.970,A 0.000,B 0.000,C -29.000}
DECL LDAT LCPDATP203={VEL 0.081,ACC 100,APO_DIST 5,APO_FAC 50.0,ORI_TYP #VAR,CIRC_TYP #BASE,JERK_FAC 50.0}
DECL FDAT FP203={TOOL_NO 2,BASE_NO 8,IPO_FRAME #BASE,POINT2[] " ",TQ_STATE FALSE}
DECL E6POS XP203={X -0.000,Y 124.070,Z -69.970,A 0.000,B 0.000,C -29.000}
DECL LDAT LCPDATP204={VEL 0.081,ACC 100,APO_DIST 5,APO_FAC 50.0,ORI_TYP #VAR,CIRC_TYP #BASE,JERK_FAC 50.0}
DECL FDAT FP204={TOOL_NO 2,BASE_NO 8,IPO_FRAME #BASE,POINT2[] " ",TQ_STATE FALSE}
DECL E6POS XP204={X -50.000,Y 124.070,Z -69.970,A 0.000,B 0.000,C -29.000}
DECL LDAT LCPDATP205={VEL 0.081,ACC 100,APO_DIST 5,APO_FAC 50.0,ORI_TYP #VAR,CIRC_TYP #BASE,JERK_FAC 50.0}
DECL FDAT FP205={TOOL_NO 2,BASE_NO 8,IPO_FRAME #BASE,POINT2[] " ",TQ_STATE FALSE}
DECL E6POS XP205={X -100.000,Y 124.070,Z -69.970,A 0.000,B 0.000,C -29.000}
DECL LDAT LCPDATP206={VEL 0.147,ACC 100,APO_DIST 5,APO_FAC 50.0,ORI_TYP #VAR,CIRC_TYP #BASE,JERK_FAC 50.0}
DECL FDAT FP206={TOOL_NO 2,BASE_NO 8,IPO_FRAME #BASE,POINT2[] " ",TQ_STATE FALSE}
DECL E6POS XP206={X -100.000,Y 170.770,Z -52.710,A 0.000,B 0.000,C -6.000}
DECL LDAT LCPDATP207={VEL 0.147,ACC 100,APO_DIST 5,APO_FAC 50.0,ORI_TYP #VAR,CIRC_TYP #BASE,JERK_FAC 50.0}
DECL FDAT FP207={TOOL_NO 2,BASE_NO 8,IPO_FRAME #BASE,POINT2[] " ",TQ_STATE FALSE}
DECL E6POS XP207={X -50.000,Y 170.770,Z -52.710,A 0.000,B 0.000,C -6.000}
DECL LDAT LCPDATP208={VEL 0.147,ACC 100,APO_DIST 5,APO_FAC 50.0,ORI_TYP #VAR,CIRC_TYP #BASE,JERK_FAC 50.0}
DECL FDAT FP208={TOOL_NO 2,BASE_NO 8,IPO_FRAME #BASE,POINT2[] " ",TQ_STATE FALSE}
DECL E6POS XP208={X -0.000,Y 170.770,Z -52.710,A 0.000,B 0.000,C -6.000}
DECL LDAT LCPDATP209={VEL 0.147,ACC 100,APO_DIST 5,APO_FAC 50.0,ORI_TYP #VAR,CIRC_TYP #BASE,JERK_FAC 50.0}
DECL FDAT FP209={TOOL_NO 2,BASE_NO 8,IPO_FRAME #BASE,POINT2[] " ",TQ_STATE FALSE}
DECL E6POS XP209={X 50.000,Y 170.770,Z -52.710,A 0.000,B 0.000,C -6.000}
DECL LDAT LCPDATP210={VEL 0.076,ACC 100,APO_DIST 5,APO_FAC 50.0,ORI_TYP #VAR,CIRC_TYP #BASE,JERK_FAC 50.0}
DECL FDAT FP210={TOOL_NO 2,BASE_NO 8,IPO_FRAME #BASE,POINT2[] " ",TQ_STATE FALSE}
DECL E6POS XP210={X 50.000,Y 145.240,Z -80.570,A 0.000,B 0.000,C -31.000}
DECL LDAT LCPDATP211={VEL 0.076,ACC 100,APO_DIST 5,APO_FAC 50.0,ORI_TYP #VAR,CIRC_TYP #BASE,JERK_FAC 50.0}
DECL FDAT FP211={TOOL_NO 2,BASE_NO 8,IPO_FRAME #BASE,POINT2[] " ",TQ_STATE FALSE}
DECL E6POS XP211={X -0.000,Y 145.240,Z -80.570,A 0.000,B 0.000,C -31.000}
DECL LDAT LCPDATP212={VEL 0.076,ACC 100,APO_DIST 5,APO_FAC 50.0,ORI_TYP #VAR,CIRC_TYP #BASE,JERK_FAC 50.0}
DECL FDAT FP212={TOOL_NO 2,BASE_NO 8,IPO_FRAME #BASE,POINT2[] " ",TQ_STATE FALSE}
DECL E6POS XP212={X -50.000,Y 145.240,Z -80.570,A 0.000,B 0.000,C -31.000}
DECL LDAT LCPDATP213={VEL 0.076,ACC 100,APO_DIST 5,APO_FAC 50.0,ORI_TYP #VAR,CIRC_TYP #BASE,JERK_FAC 50.0}
DECL FDAT FP213={TOOL_NO 2,BASE_NO 8,IPO_FRAME #BASE,POINT2[] " ",TQ_STATE FALSE}
DECL E6POS XP213={X -100.000,Y 145.240,Z -80.570,A 0.000,B 0.000,C -31.000}
DECL LDAT LCPDATP214={VEL 0.126,ACC 100,APO_DIST 5,APO_FAC 50.0,ORI_TYP #VAR,CIRC_TYP #BASE,JERK_FAC 50.0}
DECL FDAT FP214={TOOL_NO 2,BASE_NO 8,IPO_FRAME #BASE,POINT2[] " ",TQ_STATE FALSE}
DECL E6POS XP214={X -100.000,Y 168.140,Z -58.030,A 0.000,B 0.000,C -34.000}
DECL LDAT LCPDATP215={VEL 0.126,ACC 100,APO_DIST 5,APO_FAC 50.0,ORI_TYP #VAR,CIRC_TYP #BASE,JERK_FAC 50.0}
DECL FDAT FP215={TOOL_NO 2,BASE_NO 8,IPO_FRAME #BASE,POINT2[] " ",TQ_STATE FALSE}
DECL E6POS XP215={X -50.000,Y 168.140,Z -58.030,A 0.000,B 0.000,C -34.000}
DECL LDAT LCPDATP216={VEL 0.126,ACC 100,APO_DIST 5,APO_FAC 50.0,ORI_TYP #VAR,CIRC_TYP #BASE,JERK_FAC 50.0}
DECL FDAT FP216={TOOL_NO 2,BASE_NO 8,IPO_FRAME #BASE,POINT2[] " ",TQ_STATE FALSE}
DECL E6POS XP216={X -0.000,Y 168.140,Z -58.030,A 0.000,B 0.000,C -34.000}
DECL LDAT LCPDATP217={VEL 0.126,ACC 100,APO_DIST 5,APO_FAC 50.0,ORI_TYP #VAR,CIRC_TYP #BASE,JERK_FAC 50.0}
DECL FDAT FP217={TOOL_NO 2,BASE_NO 8,IPO_FRAME #BASE,POINT2[] " ",TQ_STATE FALSE}
DECL E6POS XP217={X 50.000,Y 168.140,Z -58.030,A 0.000,B 0.000,C -34.000}
DECL LDAT LCPDATP218={VEL 0.13,ACC 100,APO_DIST 5,APO_FAC 50.0,ORI_TYP #VAR,CIRC_TYP #BASE,JERK_FAC 50.0}
DECL FDAT FP218={TOOL_NO 2,BASE_NO 8,IPO_FRAME #BASE,POINT2[] " ",TQ_STATE FALSE}
DECL E6POS XP218={X 50.000,Y 200.790,Z -31.380,A 0.000,B 0.000,C -32.000}
DECL LDAT LCPDATP219={VEL 0.13,ACC 100,APO_DIST 5,APO_FAC 50.0,ORI_TYP #VAR,CIRC_TYP #BASE,JERK_FAC 50.0}
DECL FDAT FP219={TOOL_NO 2,BASE_NO 8,IPO_FRAME #BASE,POINT2[] " ",TQ_STATE FALSE}
DECL E6POS XP219={X -0.000,Y 200.790,Z -31.380,A 0.000,B 0.000,C -32.000}
DECL LDAT LCPDATP220={VEL 0.13,ACC 100,APO_DIST 5,APO_FAC 50.0,ORI_TYP #VAR,CIRC_TYP #BASE,JERK_FAC 50.0}
DECL FDAT FP220={TOOL_NO 2,BASE_NO 8,IPO_FRAME #BASE,POINT2[] " ",TQ_STATE FALSE}
DECL E6POS XP220={X -50.000,Y 200.790,Z -31.380,A 0.000,B 0.000,C -32.000}
DECL LDAT LCPDATP221={VEL 0.13,ACC 100,APO_DIST 5,APO_FAC 50.0,ORI_TYP #VAR,CIRC_TYP #BASE,JERK_FAC 50.0}
DECL FDAT FP221={TOOL_NO 2,BASE_NO 8,IPO_FRAME #BASE,POINT2[] " ",TQ_STATE FALSE}
DECL E6POS XP221={X -100.000,Y 200.790,Z -31.380,A 0.000,B 0.000,C -32.000}
DECL LDAT LCPDATP222={VEL 0.106,ACC 100,APO_DIST 5,APO_FAC 50.0,ORI_TYP #VAR,CIRC_TYP #BASE,JERK_FAC 50.0}
DECL FDAT FP222={TOOL_NO 2,BASE_NO 8,IPO_FRAME #BASE,POINT2[] " ",TQ_STATE FALSE}
DECL E6POS XP222={X -100.000,Y 225.990,Z -88.130,A 0.000,B 0.000,C -8.000}
DECL LDAT LCPDATP223={VEL 0.106,ACC 100,APO_DIST 5,APO_FAC 50.0,ORI_TYP #VAR,CIRC_TYP #BASE,JERK_FAC 50.0}
DECL FDAT FP223={TOOL_NO 2,BASE_NO 8,IPO_FRAME #BASE,POINT2[] " ",TQ_STATE FALSE}
DECL E6POS XP223={X -50.000,Y 225.990,Z -88.130,A 0.000,B 0.000,C -8.000}
DECL LDAT LCPDATP224={VEL 0.106,ACC 100,APO_DIST 5,APO_FAC 50.0,ORI_TYP #VAR,CIRC_TYP #BASE,JERK_FAC 50.0}
DECL FDAT FP224={TOOL_NO 2,BASE_NO 8,IPO_FRAME #BASE,POINT2[] " ",TQ_STATE FALSE}
DECL E6POS XP224={X -0.000,Y 225.990,Z -88.130,A 0.000,B 0.000,C -8.000}
DECL LDAT LCPDATP225={VEL 0.106,ACC 100,APO_DIST 5,APO_FAC 50.0,ORI_TYP #VAR,CIRC_TYP #BASE,JERK_FAC 50.0}
DECL FDAT FP225={TOOL_NO 2,BASE_NO 8,IPO_FRAME #BASE,POINT2[] " ",TQ_STATE FALSE}
DECL E6POS XP225={X 50.000,Y 225.990,Z -88.130,A 0.000,B 0.000,C -8.000}
DECL LDAT LCPDATP226={VEL 0.145,ACC 100,APO_DIST 5,APO_FAC 50.0,ORI_TYP #VAR,CIRC_TYP #BASE,JERK_FAC 50.0}
DECL FDAT FP226={TOOL_NO 2,BASE_NO 8,IPO_FRAME #BASE,POINT2[] " ",TQ_STATE FALSE}
DECL E6POS XP226={X 50.000,Y 209.360,Z -72.860,A 0.000,B 0.000,C -31.000}
DECL LDAT LCPDATP227={VEL 0.145,ACC 100,APO_DIST 5,APO_FAC 50.0,ORI_TYP #VAR,CIRC_TYP #BASE,JERK_FAC 50.0}
DECL FDAT FP227={TOOL_NO 2,BASE_NO 8,IPO_FRAME #BASE,POINT2[] " ",TQ_STATE FALSE}
DECL E6POS XP227={X -0.000,Y 209.360,Z -72.860,A 0.000,B 0.000,C -31.000}
DECL LDAT LCPDATP228={VEL 0.145,ACC 100,APO_DIST 5,APO_FAC 50.0,ORI_TYP #VAR,CIRC_TYP #BASE,JERK_FAC 50.0}
DECL FDAT FP228={TOOL_NO 2,BASE_NO 8,IPO_FRAME #BASE,POINT2[] " ",TQ_STATE FALSE}
DECL E6POS XP228={X -50.000,Y 209.360,Z -72.860,A 0.000,B 0.000,C -31.000}
DECL LDAT LCPDATP229={VEL 0.145,ACC 100,APO_DIST 5,APO_FAC 50.0,ORI_TYP #VAR,CIRC_TYP #BASE,JERK_FAC 50.0}
DECL FDAT FP229={TOOL_NO 2,BASE_NO 8,IPO_FRAME #BASE,POINT2[] " ",TQ_STATE FALSE}
DECL E6POS XP229={X -100.000,Y 209.360,Z -72.860,A 0.000,B 0.000,C -31.000}
DECL LDAT LCPDATP230={VEL 0.1,ACC 100,APO_DIST 5,APO_FAC 50.0,ORI_TYP #VAR,CIRC_TYP #BASE,JERK_FAC 50.0}
DECL FDAT FP230={TOOL_NO 2,BASE_NO 8,IPO_FRAME #BASE,POINT2[] " ",TQ_STATE FALSE}
DECL E6POS XP230={X -100.000,Y 244.930,Z -87.900,A 0.000,B 0.000,C -15.000}
DECL LDAT LCPDATP231={VEL 0.1,ACC 100,APO_DIST 5,APO_FAC 50.0,ORI_TYP #VAR,CIRC_TYP #BASE,JERK_FAC 50.0}
DECL FDAT FP231={TOOL_NO 2,BASE_NO 8,IPO_FRAME #BASE,POINT2[] " ",TQ_STATE FALSE}
DECL E6POS XP231={X -50.000,Y 244.930,Z -87.900,A 0.000,B 0.000,C -15.000}
DECL LDAT LCPDATP232={VEL 0.1,ACC 100,APO_DIST 5,APO_FAC 50.0,ORI_TYP #VAR,CIRC_TYP #BASE,JERK_FAC 50.0}
DECL FDAT FP232={TOOL_NO 2,BASE_NO 8,IPO_FRAME #BASE,POINT2[] " ",TQ_STATE FALSE}
DECL E6POS XP232={X -0.000,Y 244.930,Z -87.900,A 0.000,B 0.000,C -15.000}
DECL LDAT LCPDATP233={VEL 0.1,ACC 100,APO_DIST 5,APO_FAC 50.0,ORI_TYP #VAR,CIRC_TYP #BASE,JERK_FAC 50.0}
DECL FDAT FP233={TOOL_NO 2,BASE_NO 8,IPO_FRAME #BASE,POINT2[] " ",TQ_STATE FALSE}
DECL E6POS XP233={X 50.000,Y 244.930,Z -87.900,A 0.000,B 0.000,C -15.000}
DECL LDAT LCPDATP234={VEL 0.13,ACC 100,APO_DIST 5,APO_FAC 50.0,ORI_TYP #VAR,CIRC_TYP #BASE,JERK_FAC 50.0}
DECL FDAT FP234={TOOL_NO 2,BASE_NO 8,IPO_FRAME #BASE,POINT2[] " ",TQ_STATE FALSE}
DECL E6POS XP234={X 50.000,Y 261.110,Z -60.510,A 0.000,B 0.000,C -19.000}
DECL LDAT LCPDATP235={VEL 0.13,ACC 100,APO_DIST 5,APO_FAC 50.0,ORI_TYP #VAR,CIRC_TYP #BASE,JERK_FAC 50.0}
DECL FDAT FP235={TOOL_NO 2,BASE_NO 8,IPO_FRAME #BASE,POINT2[] " ",TQ_STATE FALSE}
DECL E6POS XP235={X -0.000,Y 261.110,Z -60.510,A 0.000,B 0.000,C -19.000}
DECL LDAT LCPDATP236={VEL 0.13,ACC 100,APO_DIST 5,APO_FAC 50.0,ORI_TYP #VAR,CIRC_TYP #BASE,JERK_FAC 50.0}
DECL FDAT FP236={TOOL_NO 2,BASE_NO 8,IPO_FRAME #BASE,POINT2[] " ",TQ_STATE FALSE}
DECL E6POS XP236={X -50.000,Y 261.110,Z -60.510,A 0.000,B 0.000,C -19.000}
DECL LDAT LCPDATP237={VEL 0.13,ACC 100,APO_DIST 5,APO_FAC 50.0,ORI_TYP #VAR,CIRC_TYP #BASE,JERK_FAC 50.0}
DECL FDAT FP237={TOOL_NO 2,BASE_NO 8,IPO_FRAME #BASE,POINT2[] " ",TQ_STATE FALSE}
DECL E6POS XP237={X -100.000,Y 261.110,Z -60.510,A 0.000,B 0.000,C -19.000}
DECL LDAT LCPDATP238={VEL 0.091,ACC 100,APO_DIST 5,APO_FAC 50.0,ORI_TYP #VAR,CIRC_TYP #BASE,JERK_FAC 50.0}
DECL FDAT FP238={TOOL_NO 2,BASE_NO 8,IPO_FRAME #BASE,POINT2[] " ",TQ_STATE FALSE}
DECL E6POS XP238={X -100.000,Y 287.330,Z -59.260,A 0.000,B 0.000,C -9.000}
DECL LDAT LCPDATP239={VEL 0.091,ACC 100,APO_DIST 5,APO_FAC 50.0,ORI_TYP #VAR,CIRC_TYP #BASE,JERK_FAC 50.0}
DECL FDAT FP239={TOOL_NO 2,BASE_NO 8,IPO_FRAME #BASE,POINT2[] " ",TQ_STATE FALSE}
DECL E6POS XP239={X -50.000,Y 287.330,Z -59.260,A 0.000,B 0.000,C -9.000}
DECL LDAT LCPDATP240={VEL 0.091,ACC 100,APO_DIST 5,APO_FAC 50.0,ORI_TYP #VAR,CIRC_TYP #BASE,JERK_FAC 50.0}
DECL FDAT FP240={TOOL_NO 2,BASE_NO 8,IPO_FRAME #BASE,POINT2[] " ",TQ_STATE FALSE}
DECL E6POS XP240={X -0.000,Y 287.330,Z -59.260,A 0.000,B 0.000,C -9.000}
DECL LDAT LCPDATP241={VEL 0.091,ACC 100,APO_DIST 5,APO_FAC 50.0,ORI_TYP #VAR,CIRC_TYP #BASE,JERK_FAC 50.0}
DECL FDAT FP241={TOOL_NO 2,BASE_NO 8,IPO_FRAME #BASE,POINT2[] " ",TQ_STATE FALSE}
DECL E6POS XP241={X 50.000,Y 287.330,Z -59.260,A 0.000,B 0.000,C -9.000}
DECL LDAT LCPDATP242={VEL 0.5,ACC 100,APO_DIST 5,APO_FAC 50.0,ORI_TYP #VAR,CIRC_TYP #BASE,JERK_FAC 50.0}
DECL FDAT FP242={TOOL_NO 2,BASE_NO 8,IPO_FRAME #BASE,POINT2[] " ",TQ_STATE FALSE}
DECL E6POS XP242={X 100.000,Y 296.710,Z -50.000,A 0.000,B 0.000,C 0.000}
DECL LDAT LCPDATP243={VEL 1.0,ACC 100,APO_DIST 5,APO_FAC 50.0,ORI_TYP #VAR,CIRC_TYP #BASE,JERK_FAC 50.0}
DECL FDAT FP243={TOOL_NO 2,BASE_NO 8,IPO_FRAME #BASE,POINT2[] " ",TQ_STATE FALSE}
DECL E6POS XP243={X 100.000,Y 340.000,Z -20.000,A 0.000,B 0.000,C 0.000}
DECL LDAT LCPDATP244={VEL 1.0,ACC 100,APO_DIST 5,APO_FAC 50.0,ORI_TYP #VAR,CIRC_TYP #BASE,JERK_FAC 50.0}
DECL FDAT FP244={TOOL_NO 2,BASE_NO 8,IPO_FRAME #BASE,POINT2[] " ",TQ_STATE FALSE}
DECL E6POS XP244={X 100.000,Y 340.000,Z -20.000,A 0.000,B 0.000,C 0.000}
;ENDDAT for Routine_2


; Data for Routine_3
DECL LDAT LCPDATP245={VEL 1.0,ACC 100,APO_DIST 5,APO_FAC 50.0,ORI_TYP #VAR,CIRC_TYP #BASE,JERK_FAC 50.0}
DECL FDAT FP245={TOOL_NO 2,BASE_NO 7,IPO_FRAME #BASE,POINT2[] " ",TQ_STATE FALSE}
DECL E6POS XP245={X 100.000,Y 0.000,Z -100.000,A 0.000,B 0.000,C 0.000}
DECL LDAT LCPDATP246={VEL 0.097,ACC 100,APO_DIST 5,APO_FAC 50.0,ORI_TYP #VAR,CIRC_TYP #BASE,JERK_FAC 50.0}
DECL FDAT FP246={TOOL_NO 2,BASE_NO 7,IPO_FRAME #BASE,POINT2[] " ",TQ_STATE FALSE}
DECL E6POS XP246={X 50.000,Y 7.060,Z -40.840,A 0.000,B 0.000,C -5.000}
DECL LDAT LCPDATP247={VEL 0.097,ACC 100,APO_DIST 5,APO_FAC 50.0,ORI_TYP #VAR,CIRC_TYP #BASE,JERK_FAC 50.0}
DECL FDAT FP247={TOOL_NO 2,BASE_NO 7,IPO_FRAME #BASE,POINT2[] " ",TQ_STATE FALSE}
DECL E6POS XP247={X -0.000,Y 7.060,Z -40.840,A 0.000,B 0.000,C -5.000}
DECL LDAT LCPDATP248={VEL 0.097,ACC 100,APO_DIST 5,APO_FAC 50.0,ORI_TYP #VAR,CIRC_TYP #BASE,JERK_FAC 50.0}
DECL FDAT FP248={TOOL_NO 2,BASE_NO 7,IPO_FRAME #BASE,POINT2[] " ",TQ_STATE FALSE}
DECL E6POS XP248={X -50.000,Y 7.060,Z -40.840,A 0.000,B 0.000,C -5.000}
DECL LDAT LCPDATP249={VEL 0.097,ACC 100,APO_DIST 5,APO_FAC 50.0,ORI_TYP #VAR,CIRC_TYP #BASE,JERK_FAC 50.0}
DECL FDAT FP249={TOOL_NO 2,BASE_NO 7,IPO_FRAME #BASE,POINT2[] " ",TQ_STATE FALSE}
DECL E6POS XP249={X -100.000,Y 7.060,Z -40.840,A 0.000,B 0.000,C -5.000}
DECL LDAT LCPDATP250={VEL 0.144,ACC 100,APO_DIST 5,APO_FAC 50.0,ORI_TYP #VAR,CIRC_TYP #BASE,JERK_FAC 50.0}
DECL FDAT FP250={TOOL_NO 2,BASE_NO 7,IPO_FRAME #BASE,POINT2[] " ",TQ_STATE FALSE}
DECL E6POS XP250={X -100.000,Y 5.010,Z -45.320,A 0.000,B 0.000,C -25.000}
DECL LDAT LCPDATP251={VEL 0.144,ACC 100,APO_DIST 5,APO_FAC 50.0,ORI_TYP #VAR,CIRC_TYP #BASE,JERK_FAC 50.0}
DECL FDAT FP251={TOOL_NO 2,BASE_NO 7,IPO_FRAME #BASE,POINT2[] " ",TQ_STATE FALSE}
DECL E6POS XP251={X -50.000,Y 5.010,Z -45.320,A 0.000,B 0.000,C -25.000}
DECL LDAT LCPDATP252={VEL 0.144,ACC 100,APO_DIST 5,APO_FAC 50.0,ORI_TYP #VAR,CIRC_TYP #BASE,JERK_FAC 50.0}
DECL FDAT FP252={TOOL_NO 2,BASE_NO 7,IPO_FRAME #BASE,POINT2[] " ",TQ_STATE FALSE}
DECL E6POS XP252={X -0.000,Y 5.010,Z -45.320,A 0.000,B 0.000,C -25.000}
DECL LDAT LCPDATP253={VEL 0.144,ACC 100,APO_DIST 5,APO_FAC 50.0,ORI_TYP #VAR,CIRC_TYP #BASE,JERK_FAC 50.0}
DECL FDAT FP253={TOOL_NO 2,BASE_NO 7,IPO_FRAME #BASE,POINT2[] " ",TQ_STATE FALSE}
DECL E6POS XP253={X 50.000,Y 5.010,Z -45.320,A 0.000,B 0.000,C -25.000}
DECL LDAT LCPDATP254={VEL 0.084,ACC 100,APO_DIST 5,APO_FAC 50.0,ORI_TYP #VAR,CIRC_TYP #BASE,JERK_FAC 50.0}
DECL FDAT FP254={TOOL_NO 2,BASE_NO 7,IPO_FRAME #BASE,POINT2[] " ",TQ_STATE FALSE}
DECL E6POS XP254={X 50.000,Y 26.740,Z -40.660,A 0.000,B 0.000,C -19.000}
DECL LDAT LCPDATP255={VEL 0.084,ACC 100,APO_DIST 5,APO_FAC 50.0,ORI_TYP #VAR,CIRC_TYP #BASE,JERK_FAC 50.0}
DECL FDAT FP255={TOOL_NO 2,BASE_NO 7,IPO_FRAME #BASE,POINT2[] " ",TQ_STATE FALSE}
DECL E6POS XP255={X -0.000,Y 26.740,Z -40.660,A 0.000,B 0.000,C -19.000}
DECL LDAT LCPDATP256={VEL 0.084,ACC 100,APO_DIST 5,APO_FAC 50.0,ORI_TYP #VAR,CIRC_TYP #BASE,JERK_FAC 50.0}
DECL FDAT FP256={TOOL_NO 2,BASE_NO 7,IPO_FRAME #BASE,POINT2[] " ",TQ_STATE FALSE}
DECL E6POS XP256={X -50.000,Y 26.740,Z -40.660,A 0.000,B 0.000,C -19.000}
DECL LDAT LCPDATP257={VEL 0.084,ACC 100,APO_DIST 5,APO_FAC 50.0,ORI_TYP #VAR,CIRC_TYP #BASE,JERK_FAC 50.0}
DECL FDAT FP257={TOOL_NO 2,BASE_NO 7,IPO_FRAME #BASE,POINT2[] " ",TQ_STATE FALSE}
DECL E6POS XP257={X -100.000,Y 26.740,Z -40.660,A 0.000,B 0.000,C -19.000}
DECL LDAT LCPDATP258={VEL 0.05,ACC 100,APO_DIST 5,APO_FAC 50.0,ORI_TYP #VAR,CIRC_TYP #BASE,JERK_FAC 50.0}
DECL FDAT FP258={TOOL_NO 2,BASE_NO 7,IPO_FRAME #BASE,POINT2[] " ",TQ_STATE FALSE}
DECL E6POS XP258={X -100.000,Y 19.360,Z -79.990,A 0.000,B 0.000,C -26.000}
DECL LDAT LCPDATP259={VEL 0.05,ACC 100,APO_DIST 5,APO_FAC 50.0,ORI_TYP #VAR,CIRC_TYP #BASE,JERK_FAC 50.0}
DECL FDAT FP259={TOOL_NO 2,BASE_NO 7,IPO_FRAME #BASE,POINT2[] " ",TQ_STATE FALSE}
DECL E6POS XP259={X -50.000,Y 19.360,Z -79.990,A 0.000,B 0.000,C -26.000}
DECL LDAT LCPDATP260={VEL 0.05,ACC 100,APO_DIST 5,APO_FAC 50.0,ORI_TYP #VAR,CIRC_TYP #BASE,JERK_FAC 50.0}
DECL FDAT FP260={TOOL_NO 2,BASE_NO 7,IPO_FRAME #BASE,POINT2[] " ",TQ_STATE FALSE}
DECL E6POS XP260={X -0.000,Y 19.360,Z -79.990,A 0.000,B 0.000,C -26.000}
DECL LDAT LCPDATP261={VEL 0.05,ACC 100,APO_DIST 5,APO_FAC 50.0,ORI_TYP #VAR,CIRC_TYP #BASE,JERK_FAC 50.0}
DECL FDAT FP261={TOOL_NO 2,BASE_NO 7,IPO_FRAME #BASE,POINT2[] " ",TQ_STATE FALSE}
DECL E6POS XP261={X 50.000,Y 19.360,Z -79.990,A 0.000,B 0.000,C -26.000}
DECL LDAT LCPDATP262={VEL 0.077,ACC 100,APO_DIST 5,APO_FAC 50.0,ORI_TYP #VAR,CIRC_TYP #BASE,JERK_FAC 50.0}
DECL FDAT FP262={TOOL_NO 2,BASE_NO 7,IPO_FRAME #BASE,POINT2[] " ",TQ_STATE FALSE}
DECL E6POS XP262={X 50.000,Y 64.350,Z -47.530,A 0.000,B 0.000,C -8.000}
DECL LDAT LCPDATP263={VEL 0.077,ACC 100,APO_DIST 5,APO_FAC 50.0,ORI_TYP #VAR,CIRC_TYP #BASE,JERK_FAC 50.0}
DECL FDAT FP263={TOOL_NO 2,BASE_NO 7,IPO_FRAME #BASE,POINT2[] " ",TQ_STATE FALSE}
DECL E6POS XP263={X -0.000,Y 64.350,Z -47.530,A 0.000,B 0.000,C -8.000}
DECL LDAT LCPDATP264={VEL 0.077,ACC 100,APO_DIST 5,APO_FAC 50.0,ORI_TYP #VAR,CIRC_TYP #BASE,JERK_FAC 50.0}
DECL FDAT FP264={TOOL_NO 2,BASE_NO 7,IPO_FRAME #BASE,POINT2[] " ",TQ_STATE FALSE}
DECL E6POS XP264={X -50.000,Y 64.350,Z -47.530,A 0.000,B 0.000,C -8.000}
DECL LDAT LCPDATP265={VEL 0.077,ACC 100,APO_DIST 5,APO_FAC 50.0,ORI_TYP #VAR,CIRC_TYP #BASE,JERK_FAC 50.0}
DECL FDAT FP265={TOOL_NO 2,BASE_NO 7,IPO_FRAME #BASE,POINT2[] " ",TQ_STATE FALSE}
DECL E6POS XP265={X -100.000,Y 64.350,Z -47.530,A 0.000,B 0.000,C -8.000}
DECL LDAT LCPDATP266={VEL 0.091,ACC 100,APO_DIST 5,APO_FAC 50.0,ORI_TYP #VAR,CIRC_TYP #BASE,JERK_FAC 50.0}
DECL FDAT FP266={TOOL_NO 2,BASE_NO 7,IPO_FRAME #BASE,POINT2[] " ",TQ_STATE FALSE}
DECL E6POS XP266={X -100.000,Y 33.940,Z -75.240,A 0.000,B 0.000,C -36.000}
DECL LDAT LCPDATP267={VEL 0.091,ACC 100,APO_DIST 5,APO_FAC 50.0,ORI_TYP #VAR,CIRC_TYP #BASE,JERK_FAC 50.0}
DECL FDAT FP267={TOOL_NO 2,BASE_NO 7,IPO_FRAME #BASE,POINT2[] " ",TQ_STATE FALSE}
DECL E6POS XP267={X -50.000,Y 33.940,Z -75.240,A 0.000,B 0.000,C -36.000}
DECL LDAT LCPDATP268={VEL 0.091,ACC 100,APO_DIST 5,APO_FAC 50.0,ORI_TYP #VAR,CIRC_TYP #BASE,JERK_FAC 50.0}
DECL FDAT FP268={TOOL_NO 2,BASE_NO 7,IPO_FRAME #BASE,POINT2[] " ",TQ_STATE FALSE}
DECL E6POS XP268={X -0.000,Y 33.940,Z -75.240,A 0.000,B 0.000,C -36.000}
DECL LDAT LCPDATP269={VEL 0.091,ACC 100,APO_DIST 5,APO_FAC 50.0,ORI_TYP #VAR,CIRC_TYP #BASE,JERK_FAC 50.0}
DECL FDAT FP269={TOOL_NO 2,BASE_NO 7,IPO_FRAME #BASE,POINT2[] " ",TQ_STATE FALSE}
DECL E6POS XP269={X 50.000,Y 33.940,Z -75.240,A 0.000,B 0.000,C -36.000}
DECL LDAT LCPDATP270={VEL 0.058,ACC 100,APO_DIST 5,APO_FAC 50.0,ORI_TYP #VAR,CIRC_TYP #BASE,JERK_FAC 50.0}
DECL FDAT FP270={TOOL_NO 2,BASE_NO 7,IPO_FRAME #BASE,POINT2[] " ",TQ_STATE FALSE}
DECL E6POS XP270={X 50.000,Y 90.000,Z -60.860,A 0.000,B 0.000,C -11.000}
DECL LDAT LCPDATP271={VEL 0.058,ACC 100,APO_DIST 5,APO_FAC 50.0,ORI_TYP #VAR,CIRC_TYP #BASE,JERK_FAC 50.0}
DECL FDAT FP271={TOOL_NO 2,BASE_NO 7,IPO_FRAME #BASE,POINT2[] " ",TQ_STATE FALSE}
DECL E6POS XP271={X -0.000,Y 90.000,Z -60.860,A 0.000,B 0.000,C -11.000}
DECL LDAT LCPDATP272={VEL 0.058,ACC 100,APO_DIST 5,APO_FAC 50.0,ORI_TYP #VAR,CIRC_TYP #BASE,JERK_FAC 50.0}
DECL FDAT FP272={TOOL_NO 2,BASE_NO 7,IPO_FRAME #BASE,POINT2[] " ",TQ_STATE FALSE}
DECL E6POS XP272={X -50.000,Y 90.000,Z -60.860,A 0.000,B 0.000,C -11.000}
DECL LDAT LCPDATP273={VEL 0.058,ACC 100,APO_DIST 5,APO_FAC 50.0,ORI_TYP #VAR,CIRC_TYP #BASE,JERK_FAC 50.0}
DECL FDAT FP273={TOOL_NO 2,BASE_NO 7,IPO_FRAME #BASE,POINT2[] " ",TQ_STATE FALSE}
DECL E6POS XP273={X -100.000,Y 90.000,Z -60.860,A 0.000,B 0.000,C -11.000}
DECL LDAT LCPDATP274={VEL 0.08,ACC 100,APO_DIST 5,APO_FAC 50.0,ORI_TYP #VAR,CIRC_TYP #BASE,JERK_FAC 50.0}
DECL FDAT FP274={TOOL_NO 2,BASE_NO 7,IPO_FRAME #BASE,POINT2[] " ",TQ_STATE FALSE}
DECL E6POS XP274={X -100.000,Y 108.240,Z -77.420,A 0.000,B 0.000,C -7.000}
DECL LDAT LCPDATP275={VEL 0.08,ACC 100,APO_DIST 5,APO_FAC 50.0,ORI_TYP #VAR,CIRC_TYP #BASE,JERK_FAC 50.0}
DECL FDAT FP275={TOOL_NO 2,BASE_NO 7,IPO_FRAME #BASE,POINT2[] " ",TQ_STATE FALSE}
DECL E6POS XP275={X -50.000,Y 108.240,Z -77.420,A 0.000,B 0.000,C -7.000}
DECL LDAT LCPDATP276={VEL 0.08,ACC 100,APO_DIST 5,APO_FAC 50.0,ORI_TYP #VAR,CIRC_TYP #BASE,JERK_FAC 50.0}
DECL FDAT FP276={TOOL_NO 2,BASE_NO 7,IPO_FRAME #BASE,POINT2[] " ",TQ_STATE FALSE}
DECL E6POS XP276={X -0.000,Y 108.240,Z -77.420,A 0.000,B 0.000,C -7.000}
DECL LDAT LCPDATP277={VEL 0.08,ACC 100,APO_DIST 5,APO_FAC 50.0,ORI_TYP #VAR,CIRC_TYP #BASE,JERK_FAC 50.0}
DECL FDAT FP277={TOOL_NO 2,BASE_NO 7,IPO_FRAME #BASE,POINT2[] " ",TQ_STATE FALSE}
DECL E6POS XP277={X 50.000,Y 108.240,Z -77.420,A 0.000,B 0.000,C -7.000}
DECL LDAT LCPDATP278={VEL 0.079,ACC 100,APO_DIST 5,APO_FAC 50.0,ORI_TYP #VAR,CIRC_TYP #BASE,JERK_FAC 50.0}
DECL FDAT FP278={TOOL_NO 2,BASE_NO 7,IPO_FRAME #BASE,POINT2[] " ",TQ_STATE FALSE}
DECL E6POS XP278={X 50.000,Y 111.620,Z -37.420,A 0.000,B 0.000,C -27.000}
DECL LDAT LCPDATP279={VEL 0.079,ACC 100,APO_DIST 5,APO_FAC 50.0,ORI_TYP #VAR,CIRC_TYP #BASE,JERK_FAC 50.0}
DECL FDAT FP279={TOOL_NO 2,BASE_NO 7,IPO_FRAME #BASE,POINT2[] " ",TQ_STATE FALSE}
DECL E6POS XP279={X -0.000,Y 111.620,Z -37.420,A 0.000,B 0.000,C -27.000}
DECL LDAT LCPDATP280={VEL 0.079,ACC 100,APO_DIST 5,APO_FAC 50.0,ORI_TYP #VAR,CIRC_TYP #BASE,JERK_FAC 50.0}
DECL FDAT FP280={TOOL_NO 2,BASE_NO 7,IPO_FRAME #BASE,POINT2[] " ",TQ_STATE FALSE}
DECL E6POS XP280={X -50.000,Y 111.620,Z -37.420,A 0.000,B 0.000,C -27.000}
DECL LDAT LCPDATP281={VEL 0.079,ACC 100,APO_DIST 5,APO_FAC 50.0,ORI_TYP #VAR,CIRC_TYP #BASE,JERK_FAC 50.0}
DECL FDAT FP281={TOOL_NO 2,BASE_NO 7,IPO_FRAME #BASE,POINT2[] " ",TQ_STATE FALSE}
DECL E6POS XP281={X -100.000,Y 111.620,Z -37.420,A 0.000,B 0.000,C -27.000}
DECL LDAT LCPDATP282={VEL 0.134,ACC 100,APO_DIST 5,APO_FAC 50.0,ORI_TYP #VAR,CIRC_TYP #BASE,JERK_FAC 50.0}
DECL FDAT FP282={TOOL_NO 2,BASE_NO 7,IPO_FRAME #BASE,POINT2[] " ",TQ_STATE FALSE}
DECL E6POS XP282={X -100.000,Y 124.930,Z -80.750,A 0.000,B 0.000,C -16.000}
DECL LDAT LCPDATP283={VEL 0.134,ACC 100,APO_DIST 5,APO_FAC 50.0,ORI_TYP #VAR,CIRC_TYP #BASE,JERK_FAC 50.0}
DECL FDAT FP283={TOOL_NO 2,BASE_NO 7,IPO_FRAME #BASE,POINT2[] " ",TQ_STATE FALSE}
DECL E6POS XP283={X -50.000,Y 124.930,Z -80.750,A 0.000,B 0.000,C -16.000}
DECL LDAT LCPDATP284={VEL 0.134,ACC 100,APO_DIST 5,APO_FAC 50.0,ORI_TYP #VAR,CIRC_TYP #BASE,JERK_FAC 50.0}
DECL FDAT FP284={TOOL_NO 2,BASE_NO 7,IPO_FRAME #BASE,POINT2[] " ",TQ_STATE FALSE}
DECL E6POS XP284={X -0.000,Y 124.930,Z -80.750,A 0.000,B 0.000,C -16.000}
DECL LDAT LCPDATP285={VEL 0.134,ACC 100,APO_DIST 5,APO_FAC 50.0,ORI_TYP #VAR,CIRC_TYP #BASE,JERK_FAC 50.0}
DECL FDAT FP285={TOOL_NO 2,BASE_NO 7,IPO_FRAME #BASE,POINT2[] " ",TQ_STATE FALSE}
DECL E6POS XP285={X 50.000,Y 124.930,Z -80.750,A 0.000,B 0.000,C -16.000}
DECL LDAT LCPDATP286={VEL 0.141,ACC 100,APO_DIST 5,APO_FAC 50.0,ORI_TYP #VAR,CIRC_TYP #BASE,JERK_FAC 50.0}
DECL FDAT FP286={TOOL_NO 2,BASE_NO 7,IPO_FRAME #BASE,POINT2[] " ",TQ_STATE FALSE}
DECL E6POS XP286={X 50.000,Y 137.040,Z -31.150,A 0.000,B 0.000,C -37.000}
DECL LDAT LCPDATP287={VEL 0.141,ACC 100,APO_DIST 5,APO_FAC 50.0,ORI_TYP #VAR,CIRC_TYP #BASE,JERK_FAC 50.0}
DECL FDAT FP287={TOOL_NO 2,BASE_NO 7,IPO_FRAME #BASE,POINT2[] " ",TQ_STATE FALSE}
DECL E6POS XP287={X -0.000,Y 137.040,Z -31.150,A 0.000,B 0.000,C -37.000}
DECL LDAT LCPDATP288={VEL 0.141,ACC 100,APO_DIST 5,APO_FAC 50.0,ORI_TYP #VAR,CIRC_TYP #BASE,JERK_FAC 50.0}
DECL FDAT FP288={TOOL_NO 2,BASE_NO 7,IPO_FRAME #BASE,POINT2[] " ",TQ_STATE FALSE}
DECL E6POS XP288={X -50.000,Y 137.040,Z -31.150,A 0.000,B 0.000,C -37.000}
DECL LDAT LCPDATP289={VEL 0.141,ACC 100,APO_DIST 5,APO_FAC 50.0,ORI_TYP #VAR,CIRC_TYP #BASE,JERK_FAC 50.0}
DECL FDAT FP289={TOOL_NO 2,BASE_NO 7,IPO_FRAME #BASE,POINT2[] " ",TQ_STATE FALSE}
DECL E6POS XP289={X -100.000,Y 137.040,Z -31.150,A 0.000,B 0.000,C -37.000}
DECL LDAT LCPDATP290={VEL 0.058,ACC 100,APO_DIST 5,APO_FAC 50.0,ORI_TYP #VAR,CIRC_TYP #BASE,JERK_FAC 50.0}
DECL FDAT FP290={TOOL_NO 2,BASE_NO 7,IPO_FRAME #BASE,POINT2[] " ",TQ_STATE FALSE}
DECL E6POS XP290={X -100.000,Y 144.670,Z -47.260,A 0.000,B 0.000,C -34.000}
DECL LDAT LCPDATP291={VEL 0.058,ACC 100,APO_DIST 5,APO_FAC 50.0,ORI_TYP #VAR,CIRC_TYP #BASE,JERK_FAC 50.0}
DECL FDAT FP291={TOOL_NO 2,BASE_NO 7,IPO_FRAME #BASE,POINT2[] " ",TQ_STATE FALSE}
DECL E6POS XP291={X -50.000,Y 144.670,Z -47.260,A 0.000,B 0.000,C -34.000}
DECL LDAT LCPDATP292={VEL 0.058,ACC 100,APO_DIST 5,APO_FAC 50.0,ORI_TYP #VAR,CIRC_TYP #BASE,JERK_FAC 50.0}
DECL FDAT FP292={TOOL_NO 2,BASE_NO 7,IPO_FRAME #BASE,POINT2[] " ",TQ_STATE FALSE}
DECL E6POS XP292={X -0.000,Y 144.670,Z -47.260,A 0.000,B 0.000,C -34.000}
DECL LDAT LCPDATP293={VEL 0.058,ACC 100,APO_DIST 5,APO_FAC 50.0,ORI_TYP #VAR,CIRC_TYP #BASE,JERK_FAC 50.0}
DECL FDAT FP293={TOOL_NO 2,BASE_NO 7,IPO_FRAME #BASE,POINT2[] " ",TQ_STATE FALSE}
DECL E6POS XP293={X 50.000,Y 144.670,Z -47.260,A 0.000,B 0.000,C -34.000}
DECL LDAT LCPDATP294={VEL 0.127,ACC 100,APO_DIST 5,APO_FAC 50.0,ORI_TYP #VAR,CIRC_TYP #BASE,JERK_FAC 50.0}
DECL FDAT FP294={TOOL_NO 2,BASE_NO 7,IPO_FRAME #BASE,POINT2[] " ",TQ_STATE FALSE}
DECL E6POS XP294={X 50.000,Y 175.030,Z -41.080,A 0.000,B 0.000,C -21.000}
DECL LDAT LCPDATP295={VEL 0.127,ACC 100,APO_DIST 5,APO_FAC 50.0,ORI_TYP #VAR,CIRC_TYP #BASE,JERK_FAC 50.0}
DECL FDAT FP295={TOOL_NO 2,BASE_NO 7,IPO_FRAME #BASE,POINT2[] " ",TQ_STATE FALSE}
DECL E6POS XP295={X -0.000,Y 175.030,Z -41.080,A 0.000,B 0.000,C -21.000}
DECL LDAT LCPDATP296={VEL 0.127,ACC 100,APO_DIST 5,APO_FAC 50.0,ORI_TYP #VAR,CIRC_TYP #BASE,JERK_FAC 50.0}
DECL FDAT FP296={TOOL_NO 2,BASE_NO 7,IPO_FRAME #BASE,POINT2[] " ",TQ_STATE FALSE}
DECL E6POS XP296={X -50.000,Y 175.030,Z -41.080,A 0.000,B 0.000,C -21.000}
DECL LDAT LCPDATP297={VEL 0.127,ACC 100,APO_DIST 5,APO_FAC 50.0,ORI_TYP #VAR,CIRC_TYP #BASE,JERK_FAC 50.0}
DECL FDAT FP297={TOOL_NO 2,BASE_NO 7,IPO_FRAME #BASE,POINT2[] " ",TQ_STATE FALSE}
DECL E6POS XP297={X -100.000,Y 175.030,Z -41.080,A 0.000,B 0.000,C -21.000}
DECL LDAT LCPDATP298={VEL 0.052,ACC 100,APO_DIST 5,APO_FAC 50.0,ORI_TYP #VAR,CIRC_TYP #BASE,JERK_FAC 50.0}
DECL FDAT FP298={TOOL_NO 2,BASE_NO 7,IPO_FRAME #BASE,POINT2[] " ",TQ_STATE FALSE}
DECL E6POS XP298={X -100.000,Y 200.830,Z -37.720,A 0.000,B 0.000,C -7.000}
DECL LDAT LCPDATP299={VEL 0.052,ACC 100,APO_DIST 5,APO_FAC 50.0,ORI_TYP #VAR,CIRC_TYP #BASE,JERK_FAC 50.0}
DECL FDAT FP299={TOOL_NO 2,BASE_NO 7,IPO_FRAME #BASE,POINT2[] " ",TQ_STATE FALSE}
DECL E6POS XP299={X -50.000,Y 200.830,Z -37.720,A 0.000,B 0.000,C -7.000}
DECL LDAT LCPDATP300={VEL 0.052,ACC 100,APO_DIST 5,APO_FAC 50.0,ORI_TYP #VAR,CIRC_TYP #BASE,JERK_FAC 50.0}
DECL FDAT FP300={TOOL_NO 2,BASE_NO 7,IPO_FRAME #BASE,POINT2[] " ",TQ_STATE FALSE}
DECL E6POS XP300={X -0.000,Y 200.830,Z -37.720,A 0.000,B 0.000,C -7.000}
DECL LDAT LCPDATP301={VEL 0.052,ACC 100,APO_DIST 5,APO_FAC 50.0,ORI_TYP #VAR,CIRC_TYP #BASE,JERK_FAC 50.0}
DECL FDAT FP301={TOOL_NO 2,BASE_NO 7,IPO_FRAME #BASE,POINT2[] " ",TQ_STATE FALSE}
DECL E6POS XP301={X 50.000,Y 200.830,Z -37.720,A 0.000,B 0.000,C -7.000}
DECL LDAT LCPDATP302={VEL 0.067,ACC 100,APO_DIST 5,APO_FAC 50.0,ORI_TYP #VAR,CIRC_TYP #BASE,JERK_FAC 50.0}
DECL FDAT FP302={TOOL_NO 2,BASE_NO 7,IPO_FRAME #BASE,POINT2[] " ",TQ_STATE FALSE}
DECL E6POS XP302={X 50.000,Y 192.090,Z -58.810,A 0.000,B 0.000,C -27.000}
DECL LDAT LCPDATP303={VEL 0.067,ACC 100,APO_DIST 5,APO_FAC 50.0,ORI_TYP #VAR,CIRC_TYP #BASE,JERK_FAC 50.0}
DECL FDAT FP303={TOOL_NO 2,BASE_NO 7,IPO_FRAME #BASE,POINT2[] " ",TQ_STATE FALSE}
DECL E6POS XP303={X -0.000,Y 192.090,Z -58.810,A 0.000,B 0.000,C -27.000}
DECL LDAT LCPDATP304={VEL 0.067,ACC 100,APO_DIST 5,APO_FAC 50.0,ORI_TYP #VAR,CIRC_TYP #BASE,JERK_FAC 50.0}
DECL FDAT FP304={TOOL_NO 2,BASE_NO 7,IPO_FRAME #BASE,POINT2[] " ",TQ_STATE FALSE}
DECL E6POS XP304={X -50.000,Y 192.090,Z -58.810,A 0.000,B 0.000,C -27.000}
DECL LDAT LCPDATP305={VEL 0.067,ACC 100,APO_DIST 5,APO_FAC 50.0,ORI_TYP #VAR,CIRC_TYP #BASE,JERK_FAC 50.0}
DECL FDAT FP305={TOOL_NO 2,BASE_NO 7,IPO_FRAME #BASE,POINT2[] " ",TQ_STATE FALSE}
DECL E6POS XP305={X -100.000,Y 192.090,Z -58.810,A 0.000,B 0.000,C -27.000}
DECL LDAT LCPDATP306={VEL 0.117,ACC 100,APO_DIST 5,APO_FAC 50.0,ORI_TYP #VAR,CIRC_TYP #BASE,JERK_FAC 50.0}
DECL FDAT FP306={TOOL_NO 2,BASE_NO 7,IPO_FRAME #BASE,POINT2[] " ",TQ_STATE FALSE}
DECL E6POS XP306={X -100.000,Y 235.350,Z -51.990,A 0.000,B 0.000,C -1.000}
DECL LDAT LCPDATP307={VEL 0.117,ACC 100,APO_DIST 5,APO_FAC 50.0,ORI_TYP #VAR,CIRC_TYP #BASE,JERK_FAC 50.0}
DECL FDAT FP307={TOOL_NO 2,BASE_NO 7,IPO_FRAME #BASE,POINT2[] " ",TQ_STATE FALSE}
DECL E6POS XP307={X -50.000,Y 235.350,Z -51.990,A 0.000,B 0.000,C -1.000}
DECL LDAT LCPDATP308={VEL 0.117,ACC 100,APO_DIST 5,APO_FAC 50.0,ORI_TYP #VAR,CIRC_TYP #BASE,JERK_FAC 50.0}
DECL FDAT FP308={TOOL_NO 2,BASE_NO 7,IPO_FRAME #BASE,POINT2[] " ",TQ_STATE FALSE}
DECL E6POS XP308={X -0.000,Y 235.350,Z -51.990,A 0.000,B 0.000,C -1.000}
DECL LDAT LCPDATP309={VEL 0.117,ACC 100,APO_DIST 5,APO_FAC 50.0,ORI_TYP #VAR,CIRC_TYP #BASE,JERK_FAC 50.0}
DECL FDAT FP309={TOOL_NO 2,BASE_NO 7,IPO_FRAME #BASE,POINT2[] " ",TQ_STATE FALSE}
DECL E6POS XP309={X 50.000,Y 235.350,Z -51.990,A 0.000,B 0.000,C -1.000}
DECL LDAT LCPDATP310={VEL 0.138,ACC 100,APO_DIST 5,APO_FAC 50.0,ORI_TYP #VAR,CIRC_TYP #BASE,JERK_FAC 50.0}
DECL FDAT FP310={TOOL_NO 2,BASE_NO 7,IPO_FRAME #BASE,POINT2[] " ",TQ_STATE FALSE}
DECL E6POS XP310={X 50.000,Y 230.810,Z -54.150,A 0.000,B 0.000,C -21.000}
DECL LDAT LCPDATP311={VEL 0.138,ACC 100,APO_DIST 5,APO_FAC 50.0,ORI_TYP #VAR,CIRC_TYP #BASE,JERK_FAC 50.0}
DECL FDAT FP311={TOOL_NO 2,BASE_NO 7,IPO_FRAME #BASE,POINT2[] " ",TQ_STATE FALSE}
DECL E6POS XP311={X -0.000,Y 230.810,Z -54.150,A 0.000,B 0.000,C -21.000}
DECL LDAT LCPDATP312={VEL 0.138,ACC 100,APO_DIST 5,APO_FAC 50.0,ORI_TYP #VAR,CIRC_TYP #BASE,JERK_FAC 50.0}
DECL FDAT FP312={TOOL_NO 2,BASE_NO 7,IPO_FRAME #BASE,POINT2[] " ",TQ_STATE FALSE}
DECL E6POS XP312={X -50.000,Y 230.810,Z -54.150,A 0.000,B 0.000,C -21.000}
DECL LDAT LCPDATP313={VEL 0.138,ACC 100,APO_DIST 5,APO_FAC 50.0,ORI_TYP #VAR,CIRC_TYP #BASE,JERK_FAC 50.0}
DECL FDAT FP313={TOOL_NO 2,BASE_NO 7,IPO_FRAME #BASE,POINT2[] " ",TQ_STATE FALSE}
DECL E6POS XP313={X -100.000,Y 230.810,Z -54.150,A 0.000,B 0.000,C -21.000}
DECL LDAT LCPDATP314={VEL 0.119,ACC 100,APO_DIST 5,APO_FAC 50.0,ORI_TYP #VAR,CIRC_TYP #BASE,JERK_FAC 50.0}
DECL FDAT FP314={TOOL_NO 2,BASE_NO 7,IPO_FRAME #BASE,POINT2[] " ",TQ_STATE FALSE}
DECL E6POS XP314={X -100.000,Y 263.610,Z -66.910,A 0.000,B 0.000,C -3.000}
DECL LDAT LCPDATP315={VEL 0.119,ACC 100,APO_DIST 5,APO_FAC 50.0,ORI_TYP #VAR,CIRC_TYP #BASE,JERK_FAC 50.0}
DECL FDAT FP315={TOOL_NO 2,BASE_NO 7,IPO_FRAME #BASE,POINT2[] " ",TQ_STATE FALSE}
DECL E6POS XP315={X -50.000,Y 263.610,Z -66.910,A 0.000,B 0.000,C -3.000}
DECL LDAT LCPDATP316={VEL 0.119,ACC 100,APO_DIST 5,APO_FAC 50.0,ORI_TYP #VAR,CIRC_TYP #BASE,JERK_FAC 50.0}
DECL FDAT FP316={TOOL_NO 2,BASE_NO 7,IPO_FRAME #BASE,POINT2[] " ",TQ_STATE FALSE}
DECL E6POS XP316={X -0.000,Y 263.610,Z -66.910,A 0.000,B 0.000,C -3.000}
DECL LDAT LCPDATP317={VEL 0.119,ACC 100,APO_DIST 5,APO_FAC 50.0,ORI_TYP #VAR,CIRC_TYP #BASE,JERK_FAC 50.0}
DECL FDAT FP317={TOOL_NO 2,BASE_NO 7,IPO_FRAME #BASE,POINT2[] " ",TQ_STATE FALSE}
DECL E6POS XP317={X 50.000,Y 263.610,Z -66.910,A 0.000,B 0.000,C -3.000}
DECL LDAT LCPDATP318={VEL 0.121,ACC 100,APO_DIST 5,APO_FAC 50.0,ORI_TYP #VAR,CIRC_TYP #BASE,JERK_FAC 50.0}
DECL FDAT FP318={TOOL_NO 2,BASE_NO 7,IPO_FRAME #BASE,POINT2[] " ",TQ_STATE FALSE}
DECL E6POS XP318={X 50.000,Y 261.460,Z -32.910,A 0.000,B 0.000,C -30.000}
DECL LDAT LCPDATP319={VEL 0.121,ACC 100,APO_DIST 5,APO_FAC 50.0,ORI_TYP #VAR,CIRC_TYP #BASE,JERK_FAC 50.0}
DECL FDAT FP319={TOOL_NO 2,BASE_NO 7,IPO_FRAME #BASE,POINT2[] " ",TQ_STATE FALSE}
DECL E6POS XP319={X -0.000,Y 261.460,Z -32.910,A 0.000,B 0.000,C -30.000}
DECL LDAT LCPDATP320={VEL 0.121,ACC 100,APO_DIST 5,APO_FAC 50.0,ORI_TYP #VAR,CIRC_TYP #BASE,JERK_FAC 50.0}
DECL FDAT FP320={TOOL_NO 2,BASE_NO 7,IPO_FRAME #BASE,POINT2[] " ",TQ_STATE FALSE}
DECL E6POS XP320={X -50.000,Y 261.460,Z -32.910,A 0.000,B 0.000,C -30.000}
DECL LDAT LCPDATP321={VEL 0.121,ACC 100,APO_DIST 5,APO_FAC 50.0,ORI_TYP #VAR,CIRC_TYP #BASE,JERK_FAC 50.0}
DECL FDAT FP321={TOOL_NO 2,BASE_NO 7,IPO_FRAME #BASE,POINT2[] " ",TQ_STATE FALSE}
DECL E6POS XP321={X -100.000,Y 261.460,Z -32.910,A 0.000,B 0.000,C -30.000}
DECL LDAT LCPDATP322={VEL 0.059,ACC 100,APO_DIST 5,APO_FAC 50.0,ORI_TYP #VAR,CIRC_TYP #BASE,JERK_FAC 50.0}
DECL FDAT FP322={TOOL_NO 2,BASE_NO 7,IPO_FRAME #BASE,POINT2[] " ",TQ_STATE FALSE}
DECL E6POS XP322={X -100.000,Y 274.650,Z -70.380,A 0.000,B 0.000,C -18.000}
DECL LDAT LCPDATP323={VEL 0.059,ACC 100,APO_DIST 5,APO_FAC 50.0,ORI_TYP #VAR,CIRC_TYP #BASE,JERK_FAC 50.0}
DECL FDAT FP323={TOOL_NO 2,BASE_NO 7,IPO_FRAME #BASE,POINT2[] " ",TQ_STATE FALSE}
DECL E6POS XP323={X -50.000,Y 274.650,Z -70.380,A 0.000,B 0.000,C -18.000}
DECL LDAT LCPDATP324={VEL 0.059,ACC 100,APO_DIST 5,APO_FAC 50.0,ORI_TYP #VAR,CIRC_TYP #BASE,JERK_FAC 50.0}
DECL FDAT FP324={TOOL_NO 2,BASE_NO 7,IPO_FRAME #BASE,POINT2[] " ",TQ_STATE FALSE}
DECL E6POS XP324={X -0.000,Y 274.650,Z -70.380,A 0.000,B 0.000,C -18.000}
DECL LDAT LCPDATP325={VEL 0.059,ACC 100,APO_DIST 5,APO_FAC 50.0,ORI_TYP #VAR,CIRC_TYP #BASE,JERK_FAC 50.0}
DECL FDAT FP325={TOOL_NO 2,BASE_NO 7,IPO_FRAME #BASE,POINT2[] " ",TQ_STATE FALSE}
DECL E6POS XP325={X 50.000,Y 274.650,Z -70.380,A 0.000,B 0.000,C -18.000}
DECL LDAT LCPDATP326={VEL 0.08,ACC 100,APO_DIST 5,APO_FAC 50.0,ORI_TYP #VAR,CIRC_TYP #BASE,JERK_FAC 50.0}
DECL FDAT FP326={TOOL_NO 2,BASE_NO 7,IPO_FRAME #BASE,POINT2[] " ",TQ_STATE FALSE}
DECL E6POS XP326={X 50.000,Y 276.590,Z -87.450,A 0.000,B 0.000,C -23.000}
DECL LDAT LCPDATP327={VEL 0.08,ACC 100,APO_DIST 5,APO_FAC 50.0,ORI_TYP #VAR,CIRC_TYP #BASE,JERK_FAC 50.0}
DECL FDAT FP327={TOOL_NO 2,BASE_NO 7,IPO_FRAME #BASE,POINT2[] " ",TQ_STATE FALSE}
DECL E6POS XP327={X -0.000,Y 276.590,Z -87.450,A 0.000,B 0.000,C -23.000}
DECL LDAT LCPDATP328={VEL 0.08,ACC 100,APO_DIST 5,APO_FAC 50.0,ORI_TYP #VAR,CIRC_TYP #BASE,JERK_FAC 50.0}
DECL FDAT FP328={TOOL_NO 2,BASE_NO 7,IPO_FRAME #BASE,POINT2[] " ",TQ_STATE FALSE}
DECL E6POS XP328={X -50.000,Y 276.590,Z -87.450,A 0.000,B 0.000,C -23.000}
DECL LDAT LCPDATP329={VEL 0.08,ACC 100,APO_DIST 5,APO_FAC 50.0,ORI_TYP #VAR,CIRC_TYP #BASE,JERK_FAC 50.0}
DECL FDAT FP329={TOOL_NO 2,BASE_NO 7,IPO_FRAME #BASE,POINT2[] " ",TQ_STATE FALSE}
DECL E6POS XP329={X -100.000,Y 276.590,Z -87.450,A 0.000,B 0.000,C -23.000}
DECL LDAT LCPDATP330={VEL 0.136,ACC 100,APO_DIST 5,APO_FAC 50.0,ORI_TYP #VAR,CIRC_TYP #BASE,JERK_FAC 50.0}
DECL FDAT FP330={TOOL_NO 2,BASE_NO 7,IPO_FRAME #BASE,POINT2[] " ",TQ_STATE FALSE}
DECL E6POS XP330={X -100.000,Y 311.260,Z -88.350,A 0.000,B 0.000,C -11.000}
DECL LDAT LCPDATP331={VEL 0.136,ACC 100,APO_DIST 5,APO_FAC 50.0,ORI_TYP #VAR,CIRC_TYP #BASE,JERK_FAC 50.0}
DECL FDAT FP331={TOOL_NO 2,BASE_NO 7,IPO_FRAME #BASE,POINT2[] " ",TQ_STATE FALSE}
DECL E6POS XP331={X -50.000,Y 311.260,Z -88.350,A 0.000,B 0.000,C -11.000}
DECL LDAT LCPDATP332={VEL 0.136,ACC 100,APO_DIST 5,APO_FAC 50.0,ORI_TYP #VAR,CIRC_TYP #BASE,JERK_FAC 50.0}
DECL FDAT FP332={TOOL_NO 2,BASE_NO 7,IPO_FRAME #BASE,POINT2[] " ",TQ_STATE FALSE}
DECL E6POS XP332={X -0.000,Y 311.260,Z -88.350,A 0.000,B 0.000,C -11.000}
DECL LDAT LCPDATP333={VEL 0.136,ACC 100,APO_DIST 5,APO_FAC 50.0,ORI_TYP #VAR,CIRC_TYP #BASE,JERK_FAC 50.0}
DECL FDAT FP333={TOOL_NO 2,BASE_NO 7,IPO_FRAME #BASE,POINT2[] " ",TQ_STATE FALSE}
DECL E6POS XP333={X 50.000,Y 311.260,Z -88.350,A 0.000,B 0.000,C -11.000}
DECL LDAT LCPDATP334={VEL 0.5,ACC 100,APO_DIST 5,APO_FAC 50.0,ORI_TYP #VAR,CIRC_TYP #BASE,JERK_FAC 50.0}
DECL FDAT FP334={TOOL_NO 2,BASE_NO 7,IPO_FRAME #BASE,POINT2[] " ",TQ_STATE FALSE}
DECL E6POS XP334={X 100.000,Y 328.430,Z -50.000,A 0.000,B 0.000,C 0.000}
DECL LDAT LCPDATP335={VEL 1.0,ACC 100,APO_DIST 5,APO_FAC 50.0,ORI_TYP #VAR,CIRC_TYP #BASE,JERK_FAC 50.0}
DECL FDAT FP335={TOOL_NO 2,BASE_NO 7,IPO_FRAME #BASE,POINT2[] " ",TQ_STATE FALSE}
DECL E6POS XP335={X 100.000,Y 370.000,Z -20.000,A 0.000,B 0.000,C 0.000}
DECL LDAT LCPDATP336={VEL 1.0,ACC 100,APO_DIST 5,APO_FAC 50.0,ORI_TYP #VAR,CIRC_TYP #BASE,JERK_FAC 50.0}
DECL FDAT FP336={TOOL_NO 2,BASE_NO 7,IPO_FRAME #BASE,POINT2[] " ",TQ_STATE FALSE}
DECL E6POS XP336={X 100.000,Y 370.000,Z -20.000,A 0.000,B 0.000,C 0.000}
;ENDDAT for Routine_3

ENDDAT
